RoboDK station: 4. Semi-Final Product.rdk

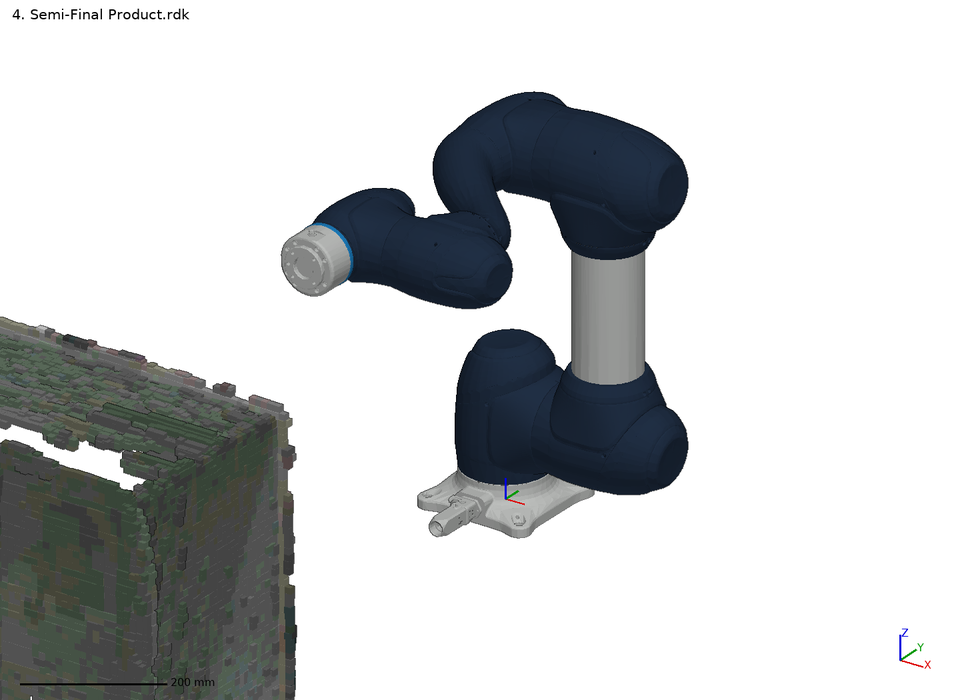
[picture v0: the station drawn from its stored meshes, robots at their saved joint values, targets as dots, program paths as lines]
Station Robotic 3D Mapping (saved by RoboDK 5.9.6). Poses are relative to the parent item; angles as X-Y-Z fixed-axis rotations.
  - frame Doosan Robotics M0609 Base at (0, 0, 0) mm
    - robot Doosan Robotics M0609: 6 axes, payload 6 kg, reach 900 mm, repeatability 0.03 mm, weight 27 kg
        modified DH rows (alpha deg, a mm, theta deg, d mm): 0, 0, 0, 135; -90, 0, -90, -6.207; 0, 411, -90, 0; -90, 0, 0, 368; 90, 0, 0, 0; -90, 0, 180, 121
        base shift (0, 0, 0) mm, rotated rx 0 ry 0 rz 180 deg
        joint limits [-360, -360, -150, -360, -360, -360] to [360, 360, 150, 360, 360, 360]; home [0, 0, 90, 0, 0, 0]; saved at [-90, 0, 90, 0, 0, 0]
      - tool Intel RealSense D455F, TCP at (0, 0, 0) mm
    - camera Camera 1
    - object Robot Base - Colored Cleaned Scan Mesh at (0, 0, 0) mm, size 1017.6 x 398.4 x 619.5 mm, geometry from 02_scan_cleaned_inside_stl_range_ROBODK_MM_COLORED.obj
  - Python program Prog1 (listed below)
  - Python program Prog2 (listed below)
  - Python program Prog3 (listed below)
  - Python program Prog4 (listed below)
  - Python program Prog5 (listed below)
  - Python program Prog6 (listed below)

--- Python program Prog1 ---
import sys
import time
from pathlib import Path

import numpy as np
import open3d as o3d
import pyrealsense2 as rs

sys.path.append("C:/RoboDK/Python")

from robodk.robolink import *
from robodk.robomath import TxyzRxyz_2_Pose, Mat


# ─────────────────────────────────────────────────────────────────────────────
# CONFIGURATION
# ─────────────────────────────────────────────────────────────────────────────

RUN_ON_REAL_ROBOT = True

HOME_JOINTS = [270.00, 0.00, 90.00, 180.00, 0.00, 0.00]

CENTER_REFERENCE_JOINTS = [270.01, 0.21, 98.95, 180.00, 6.92, 0.00]

TCP_TO_CAMERA_MOUNT = [0, 0, 55, 0, 0, 0]
CAMERA_MOUNT_TO_OPTICAL = [0, 0, 0, 0, 0, 90]

MIN_SAFE_TCP_Z_MM = 120.0
MIN_SAFE_CAMERA_Z_MM = 120.0

RS_WIDTH = 848
RS_HEIGHT = 480
RS_FPS = 30

WARMUP_FRAMES = 30
CAPTURE_FRAMES_PER_POSITION = 30

DEPTH_TRUNC_MAX = 1.0

SETTLE_TIME = 1.5
MOVE_TIMEOUT_SEC = 30.0
POLL_INTERVAL_SEC = 0.1

SURFACE_VOXEL_SIZE = 0.003

OUTLIER_NB_NEIGHBORS = 20
OUTLIER_STD_RATIO = 2.0

NORMAL_RADIUS = 0.02
NORMAL_MAX_NN = 30

SHOW_FINAL_CLOUD = True
SHOW_DEBUG_EACH_SCAN = False

MIN_SIDE_OFFSET_M = 0.08
MAX_SIDE_OFFSET_M = 0.32

MIN_VERTICAL_OFFSET_M = 0.06
MAX_VERTICAL_OFFSET_M = 0.24

MIN_FORWARD_OFFSET_M = 0.03
MAX_FORWARD_OFFSET_M = 0.14

ADAPTIVE_CROP_MARGIN_X_M = 0.12
ADAPTIVE_CROP_MARGIN_Y_M = 0.12
ADAPTIVE_CROP_MARGIN_Z_M = 0.20

BOUNDS_LOW_PERCENTILE = 2.0
BOUNDS_HIGH_PERCENTILE = 98.0

MIN_REFERENCE_POINTS = 1000

OUTPUT_FOLDER = Path(
    "C:/Users/daryl/Desktop/Robotic D Environment Mapping/"
    "Robotic-3D-Environment-Mapping/Point Cloud Testing Folder"
)

OUTPUT_CLEAN_FILE = OUTPUT_FOLDER / "adaptive_inside_box_pointcloud_clean.pcd"


# ─────────────────────────────────────────────────────────────────────────────
# ROBODK MATRIX HELPERS
# ─────────────────────────────────────────────────────────────────────────────

def robodk_mat_to_numpy(mat):
    transform = np.eye(4, dtype=np.float64)

    for row in range(3):
        for col in range(3):
            transform[row, col] = mat[row, col]

        transform[row, 3] = mat[row, 3] / 1000.0

    return transform


def numpy_to_robodk_mat(transform):
    return Mat([
        [
            transform[0, 0],
            transform[0, 1],
            transform[0, 2],
            transform[0, 3] * 1000.0,
        ],
        [
            transform[1, 0],
            transform[1, 1],
            transform[1, 2],
            transform[1, 3] * 1000.0,
        ],
        [
            transform[2, 0],
            transform[2, 1],
            transform[2, 2],
            transform[2, 3] * 1000.0,
        ],
        [0, 0, 0, 1],
    ])


def xyzrxryrz_to_numpy(pose_values):
    pose = TxyzRxyz_2_Pose([
        pose_values[0],
        pose_values[1],
        pose_values[2],
        np.radians(pose_values[3]),
        np.radians(pose_values[4]),
        np.radians(pose_values[5]),
    ])

    return robodk_mat_to_numpy(pose)


def make_local_offset_transform(offset_x, offset_y, offset_z):
    transform = np.eye(4, dtype=np.float64)
    transform[0, 3] = offset_x
    transform[1, 3] = offset_y
    transform[2, 3] = offset_z
    return transform


def joints_to_list(joints_mat):
    try:
        return list(joints_mat.list())
    except Exception:
        try:
            return list(joints_mat)
        except Exception:
            return [joints_mat[index] for index in range(len(joints_mat))]


def clamp(value, minimum_value, maximum_value):
    return max(minimum_value, min(value, maximum_value))


# ─────────────────────────────────────────────────────────────────────────────
# ROBODK ROBOT HELPERS
# ─────────────────────────────────────────────────────────────────────────────

def connect_robot(robot, rdk):
    if RUN_ON_REAL_ROBOT:
        rdk.setRunMode(RUNMODE_RUN_ROBOT)

        status = robot.ConnectSafe()
        print("ConnectSafe status:", status)

        if status != ROBOTCOM_READY:
            raise Exception("Robot is not ready. Check RoboDK connection settings.")
    else:
        rdk.setRunMode(RUNMODE_SIMULATE)
        print("Running in RoboDK simulation mode.")


def wait_until_robot_stops(robot, timeout_sec=MOVE_TIMEOUT_SEC):
    start = time.time()

    while True:
        try:
            if not robot.Busy():
                return
        except Exception:
            pass

        if time.time() - start > timeout_sec:
            raise Exception("Timeout waiting for robot to stop.")

        time.sleep(POLL_INTERVAL_SEC)


def get_robot_joints_when_ready(robot, timeout_sec=5.0):
    start = time.time()

    while True:
        try:
            return joints_to_list(robot.Joints())
        except Exception:
            if time.time() - start > timeout_sec:
                raise Exception("Could not read robot joints.")

            time.sleep(POLL_INTERVAL_SEC)


def move_robot_to_joints(robot, rdk, joints, label):
    target = rdk.AddTarget(f"_adaptive_inside_box_{label}")
    target.setAsJointTarget()
    target.setJoints(joints)

    print(f"\nMoving to {label}: {[round(joint, 2) for joint in joints]}")

    if RUN_ON_REAL_ROBOT:
        rdk.setRunMode(RUNMODE_RUN_ROBOT)
    else:
        rdk.setRunMode(RUNMODE_SIMULATE)

    robot.MoveJ(target, blocking=False)

    wait_until_robot_stops(robot)

    target.Delete()

    print(f"Arrived at {label}. Settling for {SETTLE_TIME:.1f} seconds...")
    time.sleep(SETTLE_TIME)

    return get_robot_joints_when_ready(robot)


def move_robot_to_pose(robot, rdk, T_base_tcp, label):
    target = rdk.AddTarget(f"_adaptive_inside_box_{label}")
    target_pose = numpy_to_robodk_mat(T_base_tcp)

    target.setPose(target_pose)
    target.setAsCartesianTarget()

    print(f"\nMoving to generated pose: {label}")
    print("Target TCP position in robot base frame:")
    print(f"X: {T_base_tcp[0, 3] * 1000.0:.1f} mm")
    print(f"Y: {T_base_tcp[1, 3] * 1000.0:.1f} mm")
    print(f"Z: {T_base_tcp[2, 3] * 1000.0:.1f} mm")

    if RUN_ON_REAL_ROBOT:
        rdk.setRunMode(RUNMODE_RUN_ROBOT)
    else:
        rdk.setRunMode(RUNMODE_SIMULATE)

    robot.MoveJ(target, blocking=False)

    wait_until_robot_stops(robot)

    target.Delete()

    print(f"Arrived at {label}. Settling for {SETTLE_TIME:.1f} seconds...")
    time.sleep(SETTLE_TIME)

    return get_robot_joints_when_ready(robot)


def is_generated_pose_safe(T_base_tcp, T_base_camera, label):
    tcp_z_mm = T_base_tcp[2, 3] * 1000.0
    camera_z_mm = T_base_camera[2, 3] * 1000.0

    if tcp_z_mm < MIN_SAFE_TCP_Z_MM:
        print("")
        print(f"SKIPPING {label}")
        print(f"Reason: TCP Z is too low: {tcp_z_mm:.1f} mm")
        print(f"Minimum safe TCP Z: {MIN_SAFE_TCP_Z_MM:.1f} mm")
        return False

    if camera_z_mm < MIN_SAFE_CAMERA_Z_MM:
        print("")
        print(f"SKIPPING {label}")
        print(f"Reason: Camera Z is too low: {camera_z_mm:.1f} mm")
        print(f"Minimum safe camera Z: {MIN_SAFE_CAMERA_Z_MM:.1f} mm")
        return False

    return True


def print_transform(name, transform):
    print(f"\n{name}:")
    print(np.round(transform, 6))


def print_cloud_bounds(name, point_cloud):
    if len(point_cloud.points) == 0:
        print(f"{name}: empty point cloud")
        return

    bounding_box = point_cloud.get_axis_aligned_bounding_box()

    print("")
    print(name)
    print("Points:", len(point_cloud.points))
    print("Min bound:", np.round(bounding_box.get_min_bound(), 4))
    print("Max bound:", np.round(bounding_box.get_max_bound(), 4))
    print("Center   :", np.round(bounding_box.get_center(), 4))
    print("Extent   :", np.round(bounding_box.get_extent(), 4))


# ─────────────────────────────────────────────────────────────────────────────
# REALSENSE HELPERS
# ─────────────────────────────────────────────────────────────────────────────

def start_realsense():
    print("\nStarting Intel RealSense D455f...")

    pipeline = rs.pipeline()
    config = rs.config()

    config.enable_stream(rs.stream.depth, RS_WIDTH, RS_HEIGHT, rs.format.z16, RS_FPS)
    config.enable_stream(rs.stream.color, RS_WIDTH, RS_HEIGHT, rs.format.rgb8, RS_FPS)

    profile = pipeline.start(config)

    depth_sensor = profile.get_device().first_depth_sensor()

    if depth_sensor.supports(rs.option.visual_preset):
        try:
            depth_sensor.set_option(
                rs.option.visual_preset,
                int(rs.rs400_visual_preset.high_density)
            )
            print("Visual preset: HIGH_DENSITY")
        except Exception as error:
            print("Could not set HIGH_DENSITY preset:", error)

    if depth_sensor.supports(rs.option.emitter_enabled):
        try:
            depth_sensor.set_option(rs.option.emitter_enabled, 1)
            print("Emitter enabled.")
        except Exception as error:
            print("Could not enable emitter:", error)

    if depth_sensor.supports(rs.option.laser_power):
        try:
            laser_range = depth_sensor.get_option_range(rs.option.laser_power)
            depth_sensor.set_option(rs.option.laser_power, laser_range.max)
            print("Laser power set to max:", laser_range.max)
        except Exception as error:
            print("Could not set laser power:", error)

    depth_scale = depth_sensor.get_depth_scale()
    print("Depth scale:", depth_scale)

    spatial_filter = rs.spatial_filter()
    temporal_filter = rs.temporal_filter()
    hole_filling_filter = rs.hole_filling_filter()

    spatial_filter.set_option(rs.option.filter_magnitude, 2)
    spatial_filter.set_option(rs.option.filter_smooth_alpha, 0.5)
    spatial_filter.set_option(rs.option.filter_smooth_delta, 20)

    hole_filling_filter.set_option(rs.option.holes_fill, 1)

    align = rs.align(rs.stream.color)

    print(f"Warming up RealSense for {WARMUP_FRAMES} frames...")
    for _ in range(WARMUP_FRAMES):
        pipeline.wait_for_frames()

    color_stream = profile.get_stream(rs.stream.color).as_video_stream_profile()
    intrinsics = color_stream.get_intrinsics()

    intrinsic_o3d = o3d.camera.PinholeCameraIntrinsic(
        intrinsics.width,
        intrinsics.height,
        intrinsics.fx,
        intrinsics.fy,
        intrinsics.ppx,
        intrinsics.ppy,
    )

    print(f"RealSense ready: fx={intrinsics.fx:.1f}, fy={intrinsics.fy:.1f}")

    return (
        pipeline,
        align,
        depth_scale,
        intrinsic_o3d,
        spatial_filter,
        temporal_filter,
        hole_filling_filter,
    )


def make_rgbd(color_image, depth_image, depth_scale_value):
    color_o3d = o3d.geometry.Image(color_image.astype(np.uint8))
    depth_o3d = o3d.geometry.Image(depth_image.astype(np.uint16))

    return o3d.geometry.RGBDImage.create_from_color_and_depth(
        color_o3d,
        depth_o3d,
        depth_scale=1.0 / depth_scale_value,
        depth_trunc=DEPTH_TRUNC_MAX,
        convert_rgb_to_intensity=False,
    )


def capture_stable_pointcloud(
    pipeline,
    align,
    intrinsic_o3d,
    depth_scale_value,
    spatial_filter,
    temporal_filter,
    hole_filling_filter,
    frames_to_capture=CAPTURE_FRAMES_PER_POSITION
):
    color_stack = []
    depth_stack = []

    print(f"Capturing {frames_to_capture} frames...")

    for frame_index in range(frames_to_capture):
        frames = pipeline.wait_for_frames()
        aligned_frames = align.process(frames)

        depth_frame = aligned_frames.get_depth_frame()
        color_frame = aligned_frames.get_color_frame()

        if not depth_frame or not color_frame:
            print(f"Frame {frame_index + 1}: skipped because depth or color is missing.")
            continue

        depth_frame = spatial_filter.process(depth_frame)
        depth_frame = temporal_filter.process(depth_frame)
        depth_frame = hole_filling_filter.process(depth_frame)

        depth_stack.append(np.asanyarray(depth_frame.get_data()).astype(np.uint16))
        color_stack.append(np.asanyarray(color_frame.get_data()).astype(np.uint8))

        print(f"Frame {frame_index + 1}/{frames_to_capture} captured.")

    if not depth_stack:
        return None

    print("Combining frames into one stable point cloud...")

    depth_median = np.median(np.stack(depth_stack, axis=0), axis=0).astype(np.uint16)
    color_mean = np.mean(np.stack(color_stack, axis=0), axis=0).astype(np.uint8)

    rgbd = make_rgbd(color_mean, depth_median, depth_scale_value)

    point_cloud = o3d.geometry.PointCloud.create_from_rgbd_image(
        rgbd,
        intrinsic_o3d,
    )

    if len(point_cloud.points) == 0:
        return None

    return point_cloud


# ─────────────────────────────────────────────────────────────────────────────
# ADAPTIVE POINT CLOUD HELPERS
# ─────────────────────────────────────────────────────────────────────────────

def estimate_camera_cloud_bounds(point_cloud):
    points = np.asarray(point_cloud.points)

    if len(points) < MIN_REFERENCE_POINTS:
        raise Exception(
            f"Not enough points for adaptive scan estimation. "
            f"Points found: {len(points)}"
        )

    valid_mask = (
        np.isfinite(points[:, 0]) &
        np.isfinite(points[:, 1]) &
        np.isfinite(points[:, 2]) &
        (points[:, 2] > 0.05) &
        (points[:, 2] < DEPTH_TRUNC_MAX)
    )

    points = points[valid_mask]

    if len(points) < MIN_REFERENCE_POINTS:
        raise Exception(
            f"Not enough valid depth points for adaptive scan estimation. "
            f"Valid points found: {len(points)}"
        )

    min_x = np.percentile(points[:, 0], BOUNDS_LOW_PERCENTILE)
    max_x = np.percentile(points[:, 0], BOUNDS_HIGH_PERCENTILE)

    min_y = np.percentile(points[:, 1], BOUNDS_LOW_PERCENTILE)
    max_y = np.percentile(points[:, 1], BOUNDS_HIGH_PERCENTILE)

    min_z = np.percentile(points[:, 2], BOUNDS_LOW_PERCENTILE)
    max_z = np.percentile(points[:, 2], BOUNDS_HIGH_PERCENTILE)

    center_x = float((min_x + max_x) / 2.0)
    center_y = float((min_y + max_y) / 2.0)
    center_z = float(np.median(points[:, 2]))

    extent_x = float(max_x - min_x)
    extent_y = float(max_y - min_y)
    extent_z = float(max_z - min_z)

    bounds = {
        "min_x": float(min_x),
        "max_x": float(max_x),
        "min_y": float(min_y),
        "max_y": float(max_y),
        "min_z": float(min_z),
        "max_z": float(max_z),
        "center_x": center_x,
        "center_y": center_y,
        "center_z": center_z,
        "extent_x": extent_x,
        "extent_y": extent_y,
        "extent_z": extent_z,
    }

    print("")
    print("Adaptive camera-frame bounds estimated from reference scan:")
    for key, value in bounds.items():
        print(f"{key}: {value:.4f} m")

    return bounds


def crop_pointcloud_adaptive(point_cloud, adaptive_bounds):
    if len(point_cloud.points) == 0:
        return point_cloud

    points = np.asarray(point_cloud.points)

    min_x = adaptive_bounds["min_x"] - ADAPTIVE_CROP_MARGIN_X_M
    max_x = adaptive_bounds["max_x"] + ADAPTIVE_CROP_MARGIN_X_M

    min_y = adaptive_bounds["min_y"] - ADAPTIVE_CROP_MARGIN_Y_M
    max_y = adaptive_bounds["max_y"] + ADAPTIVE_CROP_MARGIN_Y_M

    min_z = max(0.05, adaptive_bounds["min_z"] - ADAPTIVE_CROP_MARGIN_Z_M)
    max_z = min(DEPTH_TRUNC_MAX, adaptive_bounds["max_z"] + ADAPTIVE_CROP_MARGIN_Z_M)

    mask = (
        (points[:, 0] >= min_x) &
        (points[:, 0] <= max_x) &
        (points[:, 1] >= min_y) &
        (points[:, 1] <= max_y) &
        (points[:, 2] >= min_z) &
        (points[:, 2] <= max_z)
    )

    indices = np.where(mask)[0]

    if len(indices) == 0:
        print("WARNING: Adaptive crop removed all points. Keeping original cloud.")
        return point_cloud

    cropped_cloud = point_cloud.select_by_index(indices)

    print("Adaptive camera-frame crop enabled.")
    print("Points before adaptive crop:", len(point_cloud.points))
    print("Points after adaptive crop :", len(cropped_cloud.points))

    return cropped_cloud


def clean_pointcloud(point_cloud):
    if len(point_cloud.points) == 0:
        return point_cloud

    point_cloud = point_cloud.voxel_down_sample(voxel_size=SURFACE_VOXEL_SIZE)

    if len(point_cloud.points) == 0:
        return point_cloud

    point_cloud, _ = point_cloud.remove_statistical_outlier(
        nb_neighbors=OUTLIER_NB_NEIGHBORS,
        std_ratio=OUTLIER_STD_RATIO,
    )

    return point_cloud


def estimate_normals(point_cloud):
    if len(point_cloud.points) == 0:
        return point_cloud

    point_cloud.estimate_normals(
        search_param=o3d.geometry.KDTreeSearchParamHybrid(
            radius=NORMAL_RADIUS,
            max_nn=NORMAL_MAX_NN,
        )
    )

    return point_cloud


def save_debug_scan(label, point_cloud):
    debug_file = OUTPUT_FOLDER / f"debug_{label}.pcd"

    o3d.io.write_point_cloud(str(debug_file), point_cloud)

    print("Saved debug scan:", debug_file)
    print_cloud_bounds(f"Debug scan bounds - {label}", point_cloud)


# ─────────────────────────────────────────────────────────────────────────────
# ADAPTIVE SCAN POSE GENERATION
# ─────────────────────────────────────────────────────────────────────────────

def generate_adaptive_scan_offsets(adaptive_bounds):
    extent_x = adaptive_bounds["extent_x"]
    extent_y = adaptive_bounds["extent_y"]

    center_x = adaptive_bounds["center_x"]
    center_y = adaptive_bounds["center_y"]
    center_z = adaptive_bounds["center_z"]

    side_offset = clamp(
        extent_x * 0.35,
        MIN_SIDE_OFFSET_M,
        MAX_SIDE_OFFSET_M,
    )

    vertical_offset = clamp(
        extent_y * 0.35,
        MIN_VERTICAL_OFFSET_M,
        MAX_VERTICAL_OFFSET_M,
    )

    forward_offset = clamp(
        center_z * 0.12,
        MIN_FORWARD_OFFSET_M,
        MAX_FORWARD_OFFSET_M,
    )

    print("")
    print("Adaptive scan movement offsets:")
    print(f"Side offset: {side_offset:.4f} m")
    print(f"Vertical offset: {vertical_offset:.4f} m")
    print(f"Forward offset: {forward_offset:.4f} m")

    return [
        ("Reference_Center", 0.00, 0.00, 0.00),

        ("Left_Inside_Area", center_x - side_offset, center_y, 0.00),
        ("Right_Inside_Area", center_x + side_offset, center_y, 0.00),

        ("Upper_Inside_Area", center_x, center_y - vertical_offset, 0.00),
        ("Lower_Inside_Area", center_x, center_y + vertical_offset, 0.00),

        ("Upper_Left_Inside_Area", center_x - side_offset, center_y - vertical_offset, 0.00),
        ("Upper_Right_Inside_Area", center_x + side_offset, center_y - vertical_offset, 0.00),

        ("Lower_Left_Inside_Area", center_x - side_offset, center_y + vertical_offset, 0.00),
        ("Lower_Right_Inside_Area", center_x + side_offset, center_y + vertical_offset, 0.00),

        ("Closer_Center", center_x, center_y, forward_offset),
        ("Closer_Left", center_x - side_offset * 0.70, center_y, forward_offset),
        ("Closer_Right", center_x + side_offset * 0.70, center_y, forward_offset),
        ("Closer_Upper", center_x, center_y - vertical_offset * 0.70, forward_offset),
        ("Closer_Lower", center_x, center_y + vertical_offset * 0.70, forward_offset),
    ]


def generate_scan_camera_poses_from_center(T_base_camera_center, adaptive_bounds):
    generated_poses = []

    adaptive_offsets = generate_adaptive_scan_offsets(adaptive_bounds)

    print("\nGenerating adaptive scan poses from center reference...")
    print("Center camera position in robot base frame:")
    print(f"X: {T_base_camera_center[0, 3] * 1000.0:.1f} mm")
    print(f"Y: {T_base_camera_center[1, 3] * 1000.0:.1f} mm")
    print(f"Z: {T_base_camera_center[2, 3] * 1000.0:.1f} mm")

    for label, offset_x, offset_y, offset_z in adaptive_offsets:
        T_camera_offset = make_local_offset_transform(
            offset_x,
            offset_y,
            offset_z,
        )

        T_base_camera_target = T_base_camera_center @ T_camera_offset

        print("")
        print(f"Generated camera pose: {label}")
        print(f"Local offset X: {offset_x * 1000.0:.1f} mm")
        print(f"Local offset Y: {offset_y * 1000.0:.1f} mm")
        print(f"Local offset Z: {offset_z * 1000.0:.1f} mm")
        print("Generated camera position in robot base frame:")
        print(f"X: {T_base_camera_target[0, 3] * 1000.0:.1f} mm")
        print(f"Y: {T_base_camera_target[1, 3] * 1000.0:.1f} mm")
        print(f"Z: {T_base_camera_target[2, 3] * 1000.0:.1f} mm")

        generated_poses.append((label, T_base_camera_target))

    return generated_poses


# ─────────────────────────────────────────────────────────────────────────────
# SCANNING LOGIC
# ─────────────────────────────────────────────────────────────────────────────

def scan_current_position(
    label,
    pipeline,
    align,
    intrinsic_o3d,
    depth_scale,
    spatial_filter,
    temporal_filter,
    hole_filling_filter,
    T_base_camera_actual,
    adaptive_bounds=None,
):
    point_cloud = capture_stable_pointcloud(
        pipeline,
        align,
        intrinsic_o3d,
        depth_scale,
        spatial_filter,
        temporal_filter,
        hole_filling_filter,
        CAPTURE_FRAMES_PER_POSITION,
    )

    if point_cloud is None:
        print(f"WARNING: Empty point cloud at {label}.")
        return None

    print(f"Captured raw camera points at {label}: {len(point_cloud.points):,}")
    print_cloud_bounds(f"Raw camera-frame scan - {label}", point_cloud)

    if adaptive_bounds is not None:
        point_cloud = crop_pointcloud_adaptive(point_cloud, adaptive_bounds)

    if len(point_cloud.points) == 0:
        print(f"WARNING: Empty point cloud after adaptive crop at {label}.")
        return None

    print_cloud_bounds(f"Cropped camera-frame scan - {label}", point_cloud)

    point_cloud.transform(T_base_camera_actual)

    clean_scan = clean_pointcloud(point_cloud)

    if len(clean_scan.points) == 0:
        print(f"WARNING: Point cloud empty after cleaning at {label}.")
        return None

    save_debug_scan(label, clean_scan)

    if SHOW_DEBUG_EACH_SCAN:
        o3d.visualization.draw_geometries(
            [clean_scan],
            window_name=f"Debug transformed scan - {label}",
        )

    return clean_scan


# ─────────────────────────────────────────────────────────────────────────────
# MAIN
# ─────────────────────────────────────────────────────────────────────────────

def main():
    OUTPUT_FOLDER.mkdir(parents=True, exist_ok=True)

    rdk = Robolink()

    robot = rdk.ItemUserPick("Select your Doosan M0609 robot", ITEM_TYPE_ROBOT)

    if not robot.Valid():
        raise Exception("No valid robot selected.")

    print("Selected robot:", robot.Name())

    connect_robot(robot, rdk)

    T_tcp_mount = xyzrxryrz_to_numpy(TCP_TO_CAMERA_MOUNT)
    T_mount_optical = xyzrxryrz_to_numpy(CAMERA_MOUNT_TO_OPTICAL)
    T_tcp_camera = T_tcp_mount @ T_mount_optical
    T_camera_tcp = np.linalg.inv(T_tcp_camera)

    print_transform("T_tcp_camera", T_tcp_camera)

    pipeline = None
    combined_point_cloud = o3d.geometry.PointCloud()

    successful_scans = 0
    skipped_scans = 0
    unsafe_scans = 0
    failed_moves = 0

    try:
        move_robot_to_joints(
            robot,
            rdk,
            HOME_JOINTS,
            "Home_Start",
        )

        (
            pipeline,
            align,
            depth_scale,
            intrinsic_o3d,
            spatial_filter,
            temporal_filter,
            hole_filling_filter,
        ) = start_realsense()

        print("\n" + "=" * 70)
        print("ADAPTIVE INSIDE-BOX SCANNING STARTED")
        print("=" * 70)
        print("The robot moves to one manually taught center reference.")
        print("The first scan estimates the visible box size and distance.")
        print("The other scan poses are generated automatically from that estimate.")
        print("The code uses adaptive crop limits instead of a fixed 1 meter crop.")
        print("Generated poses below the robot-frame table safety limit are skipped.")
        print("=" * 70)

        center_actual_joints = move_robot_to_joints(
            robot,
            rdk,
            CENTER_REFERENCE_JOINTS,
            "Cabinet_Center_Reference",
        )

        T_base_tcp_center = robodk_mat_to_numpy(robot.SolveFK(center_actual_joints))
        T_base_camera_center = T_base_tcp_center @ T_tcp_camera

        print_transform("T_base_tcp_center", T_base_tcp_center)
        print_transform("T_base_camera_center", T_base_camera_center)

        reference_cloud = capture_stable_pointcloud(
            pipeline,
            align,
            intrinsic_o3d,
            depth_scale,
            spatial_filter,
            temporal_filter,
            hole_filling_filter,
            CAPTURE_FRAMES_PER_POSITION,
        )

        if reference_cloud is None:
            raise Exception("Reference scan failed. No point cloud was captured.")

        print_cloud_bounds("Reference raw camera-frame scan", reference_cloud)

        adaptive_bounds = estimate_camera_cloud_bounds(reference_cloud)

        reference_cloud_cropped = crop_pointcloud_adaptive(
            reference_cloud,
            adaptive_bounds,
        )

        reference_cloud_cropped.transform(T_base_camera_center)
        reference_clean_scan = clean_pointcloud(reference_cloud_cropped)

        if len(reference_clean_scan.points) > 0:
            save_debug_scan("Reference_Center", reference_clean_scan)
            combined_point_cloud += reference_clean_scan
            successful_scans += 1
            print(
                f"Accepted scan {successful_scans}: Reference_Center "
                f"with {len(reference_clean_scan.points):,} cleaned points"
            )
        else:
            print("WARNING: Reference scan became empty after cleaning.")
            skipped_scans += 1

        generated_camera_poses = generate_scan_camera_poses_from_center(
            T_base_camera_center,
            adaptive_bounds,
        )

        for label, T_base_camera_target in generated_camera_poses:
            if label == "Reference_Center":
                continue

            T_base_tcp_target = T_base_camera_target @ T_camera_tcp

            if not is_generated_pose_safe(
                T_base_tcp_target,
                T_base_camera_target,
                label,
            ):
                unsafe_scans += 1
                skipped_scans += 1
                continue

            try:
                actual_joints = move_robot_to_pose(
                    robot,
                    rdk,
                    T_base_tcp_target,
                    label,
                )
            except Exception as error:
                print("")
                print(f"WARNING: Could not move to generated pose {label}.")
                print("Move error:", error)
                failed_moves += 1
                skipped_scans += 1
                continue

            T_base_tcp_actual = robodk_mat_to_numpy(robot.SolveFK(actual_joints))
            T_base_camera_actual = T_base_tcp_actual @ T_tcp_camera

            print_transform(f"T_base_tcp_actual_{label}", T_base_tcp_actual)
            print_transform(f"T_base_camera_actual_{label}", T_base_camera_actual)

            clean_scan = scan_current_position(
                label,
                pipeline,
                align,
                intrinsic_o3d,
                depth_scale,
                spatial_filter,
                temporal_filter,
                hole_filling_filter,
                T_base_camera_actual,
                adaptive_bounds,
            )

            if clean_scan is None:
                skipped_scans += 1
                continue

            combined_point_cloud += clean_scan
            successful_scans += 1

            print(
                f"Accepted scan {successful_scans}: {label} "
                f"with {len(clean_scan.points):,} cleaned points"
            )

    except KeyboardInterrupt:
        print("\nScanning interrupted by user.")

    finally:
        if pipeline is not None:
            pipeline.stop()
            print("\nRealSense stopped.")

        try:
            move_robot_to_joints(
                robot,
                rdk,
                HOME_JOINTS,
                "Home_End",
            )
        except Exception as error:
            print("Could not move robot back to home position:", error)

    print("\n" + "=" * 70)
    print("SCAN SUMMARY")
    print("=" * 70)
    print("Successful scans:", successful_scans)
    print("Skipped scans:", skipped_scans)
    print("Unsafe skipped scans:", unsafe_scans)
    print("Failed robot moves:", failed_moves)
    print("Total merged points before final cleanup:", len(combined_point_cloud.points))
    print_cloud_bounds("Combined point cloud before final cleanup", combined_point_cloud)

    if len(combined_point_cloud.points) == 0:
        raise Exception("No valid point cloud was captured. Combined cloud is empty.")

    combined_point_cloud = clean_pointcloud(combined_point_cloud)
    combined_point_cloud = estimate_normals(combined_point_cloud)

    print("Total merged points after final cleanup:", len(combined_point_cloud.points))
    print_cloud_bounds("Combined point cloud after final cleanup", combined_point_cloud)

    o3d.io.write_point_cloud(str(OUTPUT_CLEAN_FILE), combined_point_cloud)
    print("Saved final merged point cloud to:", OUTPUT_CLEAN_FILE)

    if SHOW_FINAL_CLOUD:
        o3d.visualization.draw_geometries(
            [combined_point_cloud],
            window_name=f"Adaptive Inside Box Point Cloud - {successful_scans} scans",
        )

    print("Done.")


if __name__ == "__main__":
    main()

--- Python program Prog2 ---
import sys
from pathlib import Path

sys.path.append("C:/RoboDK/Python")

from robodk.robolink import *


ROBOTDK_EXPORT_FOLDER = Path(
    r"C:/Users/daryl/Desktop/Robotic D Environment Mapping/"
    r"Robotic-3D-Environment-Mapping/RoboDK Export"
)

COLORED_SCAN_OBJ_FILE = (
    ROBOTDK_EXPORT_FOLDER / "02_scan_cleaned_inside_stl_range_ROBODK_MM_COLORED.obj"
)

COLORED_SCAN_MTL_FILE = (
    ROBOTDK_EXPORT_FOLDER / "02_scan_cleaned_inside_stl_range_ROBODK_MM_COLORED.mtl"
)

COLORED_SCAN_PLY_FILE = (
    ROBOTDK_EXPORT_FOLDER / "02_scan_cleaned_inside_stl_range_ROBODK_MM_COLORED.ply"
)

ALIGNED_CAD_STL_FILE = (
    ROBOTDK_EXPORT_FOLDER / "04_aligned_cabinet_ROBODK_MM.stl"
)


def validate_file_exists(file_path):
    if not file_path.exists():
        raise FileNotFoundError(f"File not found: {file_path}")


def delete_existing_item(rdk, item_name):
    existing_item = rdk.Item(item_name)

    if existing_item.Valid():
        existing_item.Delete()


def import_file_to_robodk(rdk, file_path, item_name):
    validate_file_exists(file_path)

    item = rdk.AddFile(str(file_path))

    if not item.Valid():
        raise Exception(f"Could not import file into RoboDK: {file_path}")

    item.setName(item_name)
    item.setVisible(True)

    return item


def main():
    rdk = Robolink()

    scan_item_name = "Robot Base - Colored Cleaned Scan Mesh"
    cad_item_name = "Robot Base - Aligned Cabinet STL"

    delete_existing_item(rdk, scan_item_name)
    delete_existing_item(rdk, cad_item_name)

    if COLORED_SCAN_OBJ_FILE.exists():
        validate_file_exists(COLORED_SCAN_MTL_FILE)

        cleaned_scan = import_file_to_robodk(
            rdk,
            COLORED_SCAN_OBJ_FILE,
            scan_item_name
        )

        imported_scan_file = COLORED_SCAN_OBJ_FILE

    elif COLORED_SCAN_PLY_FILE.exists():
        cleaned_scan = import_file_to_robodk(
            rdk,
            COLORED_SCAN_PLY_FILE,
            scan_item_name
        )

        imported_scan_file = COLORED_SCAN_PLY_FILE

    else:
        raise FileNotFoundError(
            "No colored scan file found. Expected OBJ or PLY:\n"
            f"{COLORED_SCAN_OBJ_FILE}\n"
            f"{COLORED_SCAN_PLY_FILE}"
        )

    aligned_cad = import_file_to_robodk(
        rdk,
        ALIGNED_CAD_STL_FILE,
        cad_item_name
    )

    aligned_cad.setColor([1.0, 0.0, 0.0, 0.35])

    print("")
    print("=" * 70)
    print("IMPORTED INTO ROBODK")
    print("=" * 70)
    print("Colored scan:", cleaned_scan.Name())
    print("Scan file   :", imported_scan_file)
    print("")
    print("Aligned CAD :", aligned_cad.Name())
    print("CAD file    :", ALIGNED_CAD_STL_FILE)
    print("")
    print("The colored scan should keep its scanned color if RoboDK reads the OBJ/MTL material.")
    print("The CAD model is imported as transparent red.")
    print("Both files are already scaled to millimeters.")
    print("They should appear in the robot base coordinate position.")


if __name__ == "__main__":
    main()

--- Python program Prog3 ---
import sys
import time

import numpy as np

sys.path.append("C:/RoboDK/Python")

from robodk.robolink import *
from robodk.robomath import TxyzRxyz_2_Pose, Mat


# ─────────────────────────────────────────────────────────────────────────────
# CONFIGURATION
# ─────────────────────────────────────────────────────────────────────────────

RUN_ON_REAL_ROBOT = True

HOME_JOINTS = [270.00, 0.00, 90.00, 180.00, 0.00, 0.00]

# Your safe center camera view.
CENTER_REFERENCE_JOINTS = [270.01, 0.21, 98.95, 180.00, 6.92, 0.00]

# Your confirmed calibration. Do not change.
TCP_TO_CAMERA_MOUNT = [0, 0, 55, 0, 0, 0]
CAMERA_MOUNT_TO_OPTICAL = [0, 0, 0, 0, 0, 90]

MIN_SAFE_TCP_Z_MM = 120.0
MIN_SAFE_CAMERA_Z_MM = 120.0

SETTLE_TIME = 1.5
MOVE_TIMEOUT_SEC = 30.0
POLL_INTERVAL_SEC = 0.1

# This controls the virtual line the camera will look at.
# Think of this as the edge line inside the camera view.
#
# X = left/right in camera frame
# Y = up/down in camera frame
# Z = forward/depth in camera frame
#
# If the robot looks too far left/right, reduce LINE_HALF_WIDTH_M.
# If it looks too high/low, adjust LINE_Y_M.
# If it looks too close/far, adjust LINE_Z_M.
LINE_HALF_WIDTH_M = 0.22
LINE_Y_M = 0.06
LINE_Z_M = 0.55

# Number of look poses from left corner → center → right corner.
NUM_LOOK_POINTS = 7

# Optional small camera position offset.
# Keep these 0 first.
CAMERA_FIXED_X_OFFSET_M = 0.0
CAMERA_FIXED_Y_OFFSET_M = 0.0
CAMERA_FIXED_Z_OFFSET_M = 0.0

CREATE_DEBUG_TARGETS = True


# ─────────────────────────────────────────────────────────────────────────────
# ROBODK MATRIX HELPERS
# ─────────────────────────────────────────────────────────────────────────────

def robodk_mat_to_numpy(mat):
    transform = np.eye(4, dtype=np.float64)

    for row in range(3):
        for col in range(3):
            transform[row, col] = mat[row, col]

        transform[row, 3] = mat[row, 3] / 1000.0

    return transform


def numpy_to_robodk_mat(transform):
    return Mat([
        [
            transform[0, 0],
            transform[0, 1],
            transform[0, 2],
            transform[0, 3] * 1000.0,
        ],
        [
            transform[1, 0],
            transform[1, 1],
            transform[1, 2],
            transform[1, 3] * 1000.0,
        ],
        [
            transform[2, 0],
            transform[2, 1],
            transform[2, 2],
            transform[2, 3] * 1000.0,
        ],
        [0, 0, 0, 1],
    ])


def xyzrxryrz_to_numpy(pose_values):
    pose = TxyzRxyz_2_Pose([
        pose_values[0],
        pose_values[1],
        pose_values[2],
        np.radians(pose_values[3]),
        np.radians(pose_values[4]),
        np.radians(pose_values[5]),
    ])

    return robodk_mat_to_numpy(pose)


def joints_to_list(joints_mat):
    try:
        return list(joints_mat.list())
    except Exception:
        try:
            return list(joints_mat)
        except Exception:
            return [joints_mat[index] for index in range(len(joints_mat))]


def normalize(vector):
    norm = np.linalg.norm(vector)

    if norm < 1e-9:
        raise Exception("Cannot normalize zero-length vector.")

    return vector / norm


def print_transform(name, transform):
    print(f"\n{name}:")
    print(np.round(transform, 6))


# ─────────────────────────────────────────────────────────────────────────────
# ROBODK ROBOT HELPERS
# ─────────────────────────────────────────────────────────────────────────────

def connect_robot(robot, rdk):
    if RUN_ON_REAL_ROBOT:
        rdk.setRunMode(RUNMODE_RUN_ROBOT)

        status = robot.ConnectSafe()
        print("ConnectSafe status:", status)

        if status != ROBOTCOM_READY:
            raise Exception("Robot is not ready. Check RoboDK connection settings.")
    else:
        rdk.setRunMode(RUNMODE_SIMULATE)
        print("Running in RoboDK simulation mode.")


def wait_until_robot_stops(robot, timeout_sec=MOVE_TIMEOUT_SEC):
    start = time.time()

    while True:
        try:
            if not robot.Busy():
                return
        except Exception:
            pass

        if time.time() - start > timeout_sec:
            raise Exception("Timeout waiting for robot to stop.")

        time.sleep(POLL_INTERVAL_SEC)


def get_robot_joints_when_ready(robot, timeout_sec=5.0):
    start = time.time()

    while True:
        try:
            return joints_to_list(robot.Joints())
        except Exception:
            if time.time() - start > timeout_sec:
                raise Exception("Could not read robot joints.")

            time.sleep(POLL_INTERVAL_SEC)


def move_robot_to_joints(robot, rdk, joints, label):
    target = rdk.AddTarget(f"_camera_neck_follow_{label}")
    target.setAsJointTarget()
    target.setJoints(joints)

    print(f"\nMoving to {label}: {[round(joint, 2) for joint in joints]}")

    if RUN_ON_REAL_ROBOT:
        rdk.setRunMode(RUNMODE_RUN_ROBOT)
    else:
        rdk.setRunMode(RUNMODE_SIMULATE)

    robot.MoveJ(target, blocking=False)

    wait_until_robot_stops(robot)

    target.Delete()

    print(f"Arrived at {label}. Settling for {SETTLE_TIME:.1f} seconds...")
    time.sleep(SETTLE_TIME)

    return get_robot_joints_when_ready(robot)


def move_robot_to_pose(robot, rdk, T_base_tcp, label):
    target = rdk.AddTarget(f"_camera_neck_follow_{label}")
    target_pose = numpy_to_robodk_mat(T_base_tcp)

    target.setPose(target_pose)
    target.setAsCartesianTarget()

    print(f"\nMoving to camera neck pose: {label}")
    print("Target TCP position in robot base frame:")
    print(f"X: {T_base_tcp[0, 3] * 1000.0:.1f} mm")
    print(f"Y: {T_base_tcp[1, 3] * 1000.0:.1f} mm")
    print(f"Z: {T_base_tcp[2, 3] * 1000.0:.1f} mm")

    if RUN_ON_REAL_ROBOT:
        rdk.setRunMode(RUNMODE_RUN_ROBOT)
    else:
        rdk.setRunMode(RUNMODE_SIMULATE)

    robot.MoveJ(target, blocking=False)

    wait_until_robot_stops(robot)

    target.Delete()

    print(f"Arrived at {label}. Settling for {SETTLE_TIME:.1f} seconds...")
    time.sleep(SETTLE_TIME)

    return get_robot_joints_when_ready(robot)


def is_generated_pose_safe(T_base_tcp, T_base_camera, label):
    tcp_z_mm = T_base_tcp[2, 3] * 1000.0
    camera_z_mm = T_base_camera[2, 3] * 1000.0

    if tcp_z_mm < MIN_SAFE_TCP_Z_MM:
        print("")
        print(f"SKIPPING {label}")
        print(f"Reason: TCP Z is too low: {tcp_z_mm:.1f} mm")
        print(f"Minimum safe TCP Z: {MIN_SAFE_TCP_Z_MM:.1f} mm")
        return False

    if camera_z_mm < MIN_SAFE_CAMERA_Z_MM:
        print("")
        print(f"SKIPPING {label}")
        print(f"Reason: Camera Z is too low: {camera_z_mm:.1f} mm")
        print(f"Minimum safe camera Z: {MIN_SAFE_CAMERA_Z_MM:.1f} mm")
        return False

    return True


# ─────────────────────────────────────────────────────────────────────────────
# CAMERA LOOK / NECK MOVEMENT LOGIC
# ─────────────────────────────────────────────────────────────────────────────

def transform_point(T, point):
    point_h = np.array(
        [point[0], point[1], point[2], 1.0],
        dtype=np.float64
    )

    transformed = T @ point_h

    return transformed[:3]


def get_fixed_camera_position(T_base_camera_center):
    camera_position = T_base_camera_center[:3, 3].copy()

    camera_position += np.array([
        CAMERA_FIXED_X_OFFSET_M,
        CAMERA_FIXED_Y_OFFSET_M,
        CAMERA_FIXED_Z_OFFSET_M,
    ], dtype=np.float64)

    return camera_position


def generate_camera_frame_line_points():
    left_corner = np.array(
        [-LINE_HALF_WIDTH_M, LINE_Y_M, LINE_Z_M],
        dtype=np.float64
    )

    edge_center = np.array(
        [0.0, LINE_Y_M, LINE_Z_M],
        dtype=np.float64
    )

    right_corner = np.array(
        [LINE_HALF_WIDTH_M, LINE_Y_M, LINE_Z_M],
        dtype=np.float64
    )

    left_count = NUM_LOOK_POINTS // 2 + 1
    right_count = NUM_LOOK_POINTS - left_count + 1

    left_to_center = np.linspace(
        left_corner,
        edge_center,
        left_count
    )

    center_to_right = np.linspace(
        edge_center,
        right_corner,
        right_count
    )[1:]

    points = np.vstack((left_to_center, center_to_right))

    print("")
    print("=" * 70)
    print("Generated camera-frame look line")
    print("=" * 70)
    print("Left corner :", np.round(left_corner, 4))
    print("Edge center :", np.round(edge_center, 4))
    print("Right corner:", np.round(right_corner, 4))

    for index, point in enumerate(points, start=1):
        print(f"Look point {index:02d}: {np.round(point, 4)} m")

    return points


def transform_look_points_to_base(T_base_camera_center, camera_frame_points):
    base_points = []

    for point in camera_frame_points:
        base_point = transform_point(
            T_base_camera_center,
            point
        )

        base_points.append(base_point)

    return base_points


def build_camera_look_at_pose(
    T_base_camera_reference,
    camera_position_base,
    look_at_point_base
):
    direction = look_at_point_base - camera_position_base
    camera_forward = normalize(direction)

    reference_rotation = T_base_camera_reference[:3, :3]

    reference_up = reference_rotation[:, 1]
    reference_right = reference_rotation[:, 0]

    camera_right = np.cross(reference_up, camera_forward)

    if np.linalg.norm(camera_right) < 1e-6:
        camera_right = reference_right
    else:
        camera_right = normalize(camera_right)

    camera_up = np.cross(camera_forward, camera_right)
    camera_up = normalize(camera_up)

    camera_right = np.cross(camera_up, camera_forward)
    camera_right = normalize(camera_right)

    T_base_camera = np.eye(4, dtype=np.float64)

    T_base_camera[:3, 0] = camera_right
    T_base_camera[:3, 1] = camera_up
    T_base_camera[:3, 2] = camera_forward
    T_base_camera[:3, 3] = camera_position_base

    return T_base_camera


# ─────────────────────────────────────────────────────────────────────────────
# ROBODK DEBUG TARGETS
# ─────────────────────────────────────────────────────────────────────────────

def delete_existing_item(rdk, name, item_type):
    item = rdk.Item(name, item_type)

    if item.Valid():
        item.Delete()


def create_target_marker(rdk, name, T_base_target):
    delete_existing_item(rdk, name, ITEM_TYPE_TARGET)

    target = rdk.AddTarget(name)
    target.setPose(numpy_to_robodk_mat(T_base_target))

    return target


def create_point_marker(rdk, name, position_base):
    T_base_target = np.eye(4, dtype=np.float64)
    T_base_target[:3, 3] = position_base

    return create_target_marker(
        rdk,
        name,
        T_base_target
    )


def create_debug_targets(
    rdk,
    look_points_base,
    camera_position_base,
    camera_pose_targets
):
    if not CREATE_DEBUG_TARGETS:
        return

    create_point_marker(
        rdk,
        "NECK_CAMERA_FIXED_POSITION",
        camera_position_base
    )

    for index, look_point in enumerate(look_points_base, start=1):
        create_point_marker(
            rdk,
            f"NECK_LOOK_POINT_{index:02d}",
            look_point
        )

    for index, T_base_tcp in enumerate(camera_pose_targets, start=1):
        create_target_marker(
            rdk,
            f"NECK_TCP_TARGET_{index:02d}",
            T_base_tcp
        )


# ─────────────────────────────────────────────────────────────────────────────
# MAIN
# ─────────────────────────────────────────────────────────────────────────────

def main():
    rdk = Robolink()

    robot = rdk.ItemUserPick(
        "Select your Doosan M0609 robot",
        ITEM_TYPE_ROBOT
    )

    if not robot.Valid():
        raise Exception("No valid robot selected.")

    print("Selected robot:", robot.Name())

    connect_robot(robot, rdk)

    T_tcp_mount = xyzrxryrz_to_numpy(TCP_TO_CAMERA_MOUNT)
    T_mount_optical = xyzrxryrz_to_numpy(CAMERA_MOUNT_TO_OPTICAL)

    T_tcp_camera = T_tcp_mount @ T_mount_optical
    T_camera_tcp = np.linalg.inv(T_tcp_camera)

    print_transform("T_tcp_camera", T_tcp_camera)

    try:
        move_robot_to_joints(
            robot,
            rdk,
            HOME_JOINTS,
            "Home_Start"
        )

        center_actual_joints = move_robot_to_joints(
            robot,
            rdk,
            CENTER_REFERENCE_JOINTS,
            "Center_Reference_View"
        )

        T_base_tcp_center = robodk_mat_to_numpy(
            robot.SolveFK(center_actual_joints)
        )

        T_base_camera_center = T_base_tcp_center @ T_tcp_camera

        print_transform("T_base_tcp_center", T_base_tcp_center)
        print_transform("T_base_camera_center", T_base_camera_center)

        camera_frame_look_points = generate_camera_frame_line_points()

        look_points_base = transform_look_points_to_base(
            T_base_camera_center,
            camera_frame_look_points
        )

        fixed_camera_position_base = get_fixed_camera_position(
            T_base_camera_center
        )

        camera_pose_targets = []

        print("")
        print("=" * 70)
        print("GENERATING CAMERA NECK FOLLOW POSES")
        print("=" * 70)
        print("Camera position stays fixed.")
        print("Only the camera orientation changes.")
        print("Motion: left corner → edge center → right corner.")
        print("=" * 70)

        for index, look_point_base in enumerate(look_points_base, start=1):
            label = f"Neck_Follow_Point_{index:02d}"

            print("")
            print(label)
            print("Camera fixed position:")
            print(np.round(fixed_camera_position_base * 1000.0, 2), "mm")
            print("Looking at:")
            print(np.round(look_point_base * 1000.0, 2), "mm")

            T_base_camera_look = build_camera_look_at_pose(
                T_base_camera_center,
                fixed_camera_position_base,
                look_point_base
            )

            T_base_tcp_look = T_base_camera_look @ T_camera_tcp

            camera_pose_targets.append(T_base_tcp_look)

            if not is_generated_pose_safe(
                T_base_tcp_look,
                T_base_camera_look,
                label
            ):
                continue

        create_debug_targets(
            rdk,
            look_points_base,
            fixed_camera_position_base,
            camera_pose_targets
        )

        print("")
        print("=" * 70)
        print("CAMERA NECK FOLLOW START")
        print("=" * 70)

        for index, T_base_tcp_target in enumerate(camera_pose_targets, start=1):
            label = f"Neck_Follow_Point_{index:02d}"

            move_robot_to_pose(
                robot,
                rdk,
                T_base_tcp_target,
                label
            )

        print("")
        print("=" * 70)
        print("CAMERA NECK FOLLOW FINISHED")
        print("=" * 70)

    except KeyboardInterrupt:
        print("")
        print("Movement interrupted by user.")

    finally:
        try:
            move_robot_to_joints(
                robot,
                rdk,
                HOME_JOINTS,
                "Home_End"
            )
        except Exception as error:
            print("Could not move robot back to home position:", error)

    print("Done.")


if __name__ == "__main__":
    main()

--- Python program Prog4 ---
import sys
import time

import numpy as np

sys.path.append("C:/RoboDK/Python")

from robodk.robolink import *
from robodk.robomath import TxyzRxyz_2_Pose, Mat


# ─────────────────────────────────────────────────────────────────────────────
# CONFIGURATION
# ─────────────────────────────────────────────────────────────────────────────

RUN_ON_REAL_ROBOT = True

HOME_JOINTS = [270.00, 0.00, 90.00, 180.00, 0.00, 0.00]

CENTER_REFERENCE_JOINTS = [270.01, 0.21, 98.95, 180.00, 6.92, 0.00]

# Existing sensor/camera calibration.
TCP_TO_CAMERA_MOUNT = [0, 0, 55, 0, 0, 0]
CAMERA_MOUNT_TO_OPTICAL = [0, 0, 0, 0, 0, 90]

MIN_SAFE_TCP_Z_MM = 120.0

SETTLE_TIME = 1.5
MOVE_TIMEOUT_SEC = 30.0
POLL_INTERVAL_SEC = 0.1

# The seam is defined in the camera frame.
# X = left/right
# Y = up/down
# Z = forward/depth
#
# Previous values were too far. These are closer and safer.
SEAM_HALF_WIDTH_M = 0.08
SEAM_Y_M = 0.06
SEAM_Z_M = 0.18

# Keeps the dry-run tip slightly above the imagined seam.
DRY_RUN_HEIGHT_OFFSET_M = 0.03

# Distance before the seam along the torch direction.
# Smaller = tip gets nearer to the edge.
TIP_STANDOFF_M = 0.02

NUM_PATH_POINTS = 5

# Keep J6 close to the center value, but allow RoboDK to solve IK.
LOCK_J6_WITH_SEED = True
MAX_J6_WARNING_DEGREES = 5.0

CREATE_DEBUG_TARGETS = True


# ─────────────────────────────────────────────────────────────────────────────
# MATRIX HELPERS
# ─────────────────────────────────────────────────────────────────────────────

def robodk_mat_to_numpy(mat):
    transform = np.eye(4, dtype=np.float64)

    for row in range(3):
        for col in range(3):
            transform[row, col] = mat[row, col]

        transform[row, 3] = mat[row, 3] / 1000.0

    return transform


def numpy_to_robodk_mat(transform):
    return Mat([
        [
            transform[0, 0],
            transform[0, 1],
            transform[0, 2],
            transform[0, 3] * 1000.0,
        ],
        [
            transform[1, 0],
            transform[1, 1],
            transform[1, 2],
            transform[1, 3] * 1000.0,
        ],
        [
            transform[2, 0],
            transform[2, 1],
            transform[2, 2],
            transform[2, 3] * 1000.0,
        ],
        [0, 0, 0, 1],
    ])


def xyzrxryrz_to_numpy(pose_values):
    pose = TxyzRxyz_2_Pose([
        pose_values[0],
        pose_values[1],
        pose_values[2],
        np.radians(pose_values[3]),
        np.radians(pose_values[4]),
        np.radians(pose_values[5]),
    ])

    return robodk_mat_to_numpy(pose)


def joints_to_list(joints_mat):
    try:
        return list(joints_mat.list())
    except Exception:
        try:
            return list(joints_mat)
        except Exception:
            return [joints_mat[index] for index in range(len(joints_mat))]


def normalize(vector):
    norm = np.linalg.norm(vector)

    if norm < 1e-9:
        raise Exception("Cannot normalize zero-length vector.")

    return vector / norm


def transform_point(transform, point):
    point_h = np.array(
        [point[0], point[1], point[2], 1.0],
        dtype=np.float64
    )

    transformed = transform @ point_h

    return transformed[:3]


def print_transform(name, transform):
    print(f"\n{name}:")
    print(np.round(transform, 6))


# ─────────────────────────────────────────────────────────────────────────────
# ROBOT HELPERS
# ─────────────────────────────────────────────────────────────────────────────

def connect_robot(robot, rdk):
    if RUN_ON_REAL_ROBOT:
        rdk.setRunMode(RUNMODE_RUN_ROBOT)

        status = robot.ConnectSafe()
        print("ConnectSafe status:", status)

        if status != ROBOTCOM_READY:
            raise Exception("Robot is not ready. Check RoboDK connection settings.")
    else:
        rdk.setRunMode(RUNMODE_SIMULATE)
        print("Running in RoboDK simulation mode.")


def wait_until_robot_stops(robot, timeout_sec=MOVE_TIMEOUT_SEC):
    start = time.time()

    while True:
        try:
            if not robot.Busy():
                return
        except Exception:
            pass

        if time.time() - start > timeout_sec:
            raise Exception("Timeout waiting for robot to stop.")

        time.sleep(POLL_INTERVAL_SEC)


def get_robot_joints_when_ready(robot, timeout_sec=5.0):
    start = time.time()

    while True:
        try:
            return joints_to_list(robot.Joints())
        except Exception:
            if time.time() - start > timeout_sec:
                raise Exception("Could not read robot joints.")

            time.sleep(POLL_INTERVAL_SEC)


def move_robot_to_joints(robot, rdk, joints, label):
    target = rdk.AddTarget(f"_angled_tip_path_{label}")
    target.setAsJointTarget()
    target.setJoints(joints)

    print(f"\nMoving to {label}: {[round(joint, 2) for joint in joints]}")

    if RUN_ON_REAL_ROBOT:
        rdk.setRunMode(RUNMODE_RUN_ROBOT)
    else:
        rdk.setRunMode(RUNMODE_SIMULATE)

    robot.MoveJ(target, blocking=False)

    wait_until_robot_stops(robot)

    target.Delete()

    print(f"Arrived at {label}. Settling for {SETTLE_TIME:.1f} seconds...")
    time.sleep(SETTLE_TIME)

    return get_robot_joints_when_ready(robot)


def move_robot_to_pose(
    robot,
    rdk,
    T_base_tcp,
    seed_joints,
    locked_j6_value,
    label
):
    target = rdk.AddTarget(f"_angled_tip_path_{label}")
    target_pose = numpy_to_robodk_mat(T_base_tcp)

    target.setPose(target_pose)
    target.setAsCartesianTarget()

    seed = list(seed_joints)

    if LOCK_J6_WITH_SEED:
        seed[5] = locked_j6_value

    target.setJoints(seed)

    print(f"\nMoving to angled tip pose: {label}")
    print("Target TCP position in robot base frame:")
    print(f"X: {T_base_tcp[0, 3] * 1000.0:.1f} mm")
    print(f"Y: {T_base_tcp[1, 3] * 1000.0:.1f} mm")
    print(f"Z: {T_base_tcp[2, 3] * 1000.0:.1f} mm")
    print("Seed joints:")
    print([round(joint, 2) for joint in seed])

    if RUN_ON_REAL_ROBOT:
        rdk.setRunMode(RUNMODE_RUN_ROBOT)
    else:
        rdk.setRunMode(RUNMODE_SIMULATE)

    robot.MoveJ(target, blocking=False)

    wait_until_robot_stops(robot)

    actual_joints = get_robot_joints_when_ready(robot)

    target.Delete()

    print(f"Arrived at {label}. Settling for {SETTLE_TIME:.1f} seconds...")
    print("Actual joints:")
    print([round(joint, 2) for joint in actual_joints])
    print("Actual J6:", round(actual_joints[5], 2))

    if abs(actual_joints[5] - locked_j6_value) > MAX_J6_WARNING_DEGREES:
        print("")
        print("WARNING: J6 changed more than expected.")
        print("The angle may require a different wrist configuration.")

    time.sleep(SETTLE_TIME)

    return actual_joints


def is_pose_safe(T_base_tcp, label):
    tcp_z_mm = T_base_tcp[2, 3] * 1000.0

    if tcp_z_mm < MIN_SAFE_TCP_Z_MM:
        print("")
        print(f"SKIPPING {label}")
        print(f"Reason: TCP Z is too low: {tcp_z_mm:.1f} mm")
        return False

    return True


# ─────────────────────────────────────────────────────────────────────────────
# SEAM PATH GENERATION
# ─────────────────────────────────────────────────────────────────────────────

def generate_seam_points_camera_frame():
    left_corner = np.array(
        [
            -SEAM_HALF_WIDTH_M,
            SEAM_Y_M + DRY_RUN_HEIGHT_OFFSET_M,
            SEAM_Z_M
        ],
        dtype=np.float64
    )

    center_edge = np.array(
        [
            0.0,
            SEAM_Y_M + DRY_RUN_HEIGHT_OFFSET_M,
            SEAM_Z_M
        ],
        dtype=np.float64
    )

    right_corner = np.array(
        [
            SEAM_HALF_WIDTH_M,
            SEAM_Y_M + DRY_RUN_HEIGHT_OFFSET_M,
            SEAM_Z_M
        ],
        dtype=np.float64
    )

    left_count = NUM_PATH_POINTS // 2 + 1
    right_count = NUM_PATH_POINTS - left_count + 1

    left_to_center = np.linspace(
        left_corner,
        center_edge,
        left_count
    )

    center_to_right = np.linspace(
        center_edge,
        right_corner,
        right_count
    )[1:]

    points = np.vstack((left_to_center, center_to_right))

    print("")
    print("=" * 70)
    print("Generated angled seam points in camera frame")
    print("=" * 70)
    print("Left corner :", np.round(left_corner, 4))
    print("Center edge :", np.round(center_edge, 4))
    print("Right corner:", np.round(right_corner, 4))

    for index, point in enumerate(points, start=1):
        print(f"Seam point {index:02d}: {np.round(point, 4)} m")

    return points


def transform_seam_points_to_base(T_base_camera_center, seam_points_camera):
    seam_points_base = []

    for point in seam_points_camera:
        seam_points_base.append(
            transform_point(
                T_base_camera_center,
                point
            )
        )

    return seam_points_base


# ─────────────────────────────────────────────────────────────────────────────
# ANGLED TOOL FRAME
# ─────────────────────────────────────────────────────────────────────────────

def build_angled_tcp_pose(
    camera_position_base,
    seam_point_base,
    seam_direction_base,
    reference_rotation
):
    # Tool points from robot/camera side toward the seam.
    # This is the missing "angle where it is looking at".
    approach_axis = normalize(seam_point_base - camera_position_base)

    # Keep X roughly along the welding seam.
    tool_x_axis = seam_direction_base - np.dot(seam_direction_base, approach_axis) * approach_axis

    if np.linalg.norm(tool_x_axis) < 1e-6:
        tool_x_axis = reference_rotation[:, 0]
    else:
        tool_x_axis = normalize(tool_x_axis)

    # Build a clean right-handed orientation.
    tool_y_axis = np.cross(approach_axis, tool_x_axis)
    tool_y_axis = normalize(tool_y_axis)

    tool_x_axis = np.cross(tool_y_axis, approach_axis)
    tool_x_axis = normalize(tool_x_axis)

    # Keep the TCP slightly before the seam, so the tip is close but not too far in.
    tcp_position = seam_point_base - approach_axis * TIP_STANDOFF_M

    T_base_tcp = np.eye(4, dtype=np.float64)
    T_base_tcp[:3, 0] = tool_x_axis
    T_base_tcp[:3, 1] = tool_y_axis
    T_base_tcp[:3, 2] = approach_axis
    T_base_tcp[:3, 3] = tcp_position

    return T_base_tcp


def generate_angled_tcp_targets(
    T_base_camera_center,
    seam_points_base
):
    if len(seam_points_base) < 2:
        raise Exception("Not enough seam points.")

    camera_position_base = T_base_camera_center[:3, 3]
    reference_rotation = T_base_camera_center[:3, :3]

    seam_direction_base = seam_points_base[-1] - seam_points_base[0]
    seam_direction_base = normalize(seam_direction_base)

    targets = []

    print("")
    print("=" * 70)
    print("Generating angled TCP targets")
    print("=" * 70)
    print("The tool now points toward the seam.")
    print("The tip is closer because of TIP_STANDOFF_M.")

    for index, seam_point_base in enumerate(seam_points_base, start=1):
        label = f"Angled_Tip_Point_{index:02d}"

        T_base_tcp = build_angled_tcp_pose(
            camera_position_base,
            seam_point_base,
            seam_direction_base,
            reference_rotation
        )

        targets.append(
            (
                label,
                T_base_tcp,
                seam_point_base
            )
        )

        print("")
        print(label)
        print("Seam point:")
        print(np.round(seam_point_base * 1000.0, 2), "mm")
        print("TCP point:")
        print(np.round(T_base_tcp[:3, 3] * 1000.0, 2), "mm")
        print("Tool approach direction:")
        print(np.round(T_base_tcp[:3, 2], 4))

    return targets


# ─────────────────────────────────────────────────────────────────────────────
# DEBUG TARGETS
# ─────────────────────────────────────────────────────────────────────────────

def delete_existing_item(rdk, name, item_type):
    item = rdk.Item(name, item_type)

    if item.Valid():
        item.Delete()


def create_target_marker(rdk, name, T_base_target):
    if not CREATE_DEBUG_TARGETS:
        return None

    delete_existing_item(rdk, name, ITEM_TYPE_TARGET)

    target = rdk.AddTarget(name)
    target.setPose(numpy_to_robodk_mat(T_base_target))

    return target


def create_point_marker(rdk, name, position_base):
    T_base_target = np.eye(4, dtype=np.float64)
    T_base_target[:3, 3] = position_base

    return create_target_marker(
        rdk,
        name,
        T_base_target
    )


def create_debug_targets(rdk, targets):
    if not CREATE_DEBUG_TARGETS:
        return

    for index, (_, T_base_tcp, seam_point_base) in enumerate(targets, start=1):
        create_target_marker(
            rdk,
            f"ANGLED_TCP_TARGET_{index:02d}",
            T_base_tcp
        )

        create_point_marker(
            rdk,
            f"ANGLED_SEAM_POINT_{index:02d}",
            seam_point_base
        )


# ─────────────────────────────────────────────────────────────────────────────
# MAIN
# ─────────────────────────────────────────────────────────────────────────────

def main():
    rdk = Robolink()

    robot = rdk.ItemUserPick(
        "Select your Doosan M0609 robot",
        ITEM_TYPE_ROBOT
    )

    if not robot.Valid():
        raise Exception("No valid robot selected.")

    print("Selected robot:", robot.Name())

    connect_robot(robot, rdk)

    T_tcp_mount = xyzrxryrz_to_numpy(TCP_TO_CAMERA_MOUNT)
    T_mount_optical = xyzrxryrz_to_numpy(CAMERA_MOUNT_TO_OPTICAL)

    T_tcp_camera = T_tcp_mount @ T_mount_optical

    print_transform("T_tcp_camera", T_tcp_camera)

    try:
        move_robot_to_joints(
            robot,
            rdk,
            HOME_JOINTS,
            "Home_Start"
        )

        actual_center_joints = move_robot_to_joints(
            robot,
            rdk,
            CENTER_REFERENCE_JOINTS,
            "Center_Reference_View"
        )

        locked_j6_value = actual_center_joints[5]

        T_base_tcp_center = robodk_mat_to_numpy(
            robot.SolveFK(actual_center_joints)
        )

        T_base_camera_center = T_base_tcp_center @ T_tcp_camera

        print_transform("T_base_tcp_center", T_base_tcp_center)
        print_transform("T_base_camera_center", T_base_camera_center)
        print("")
        print("J6 reference value:", round(locked_j6_value, 2))

        seam_points_camera = generate_seam_points_camera_frame()

        seam_points_base = transform_seam_points_to_base(
            T_base_camera_center,
            seam_points_camera
        )

        targets = generate_angled_tcp_targets(
            T_base_camera_center,
            seam_points_base
        )

        create_debug_targets(
            rdk,
            targets
        )

        print("")
        print("=" * 70)
        print("ANGLED TIP PATH START")
        print("=" * 70)
        print("The tool now has an angle toward the seam.")
        print("The TCP is placed slightly before the seam using TIP_STANDOFF_M.")
        print("No welding machine or arc is triggered.")
        print("=" * 70)

        successful_moves = 0
        skipped_moves = 0
        failed_moves = 0

        seed_joints = actual_center_joints

        for label, T_base_tcp_target, seam_point_base in targets:
            if not is_pose_safe(
                T_base_tcp_target,
                label
            ):
                skipped_moves += 1
                continue

            try:
                actual_joints = move_robot_to_pose(
                    robot,
                    rdk,
                    T_base_tcp_target,
                    seed_joints,
                    locked_j6_value,
                    label
                )

                if LOCK_J6_WITH_SEED:
                    actual_joints[5] = locked_j6_value

                seed_joints = actual_joints

                successful_moves += 1

            except Exception as error:
                print("")
                print(f"WARNING: Could not move to {label}.")
                print("Move error:", error)
                failed_moves += 1
                continue

        print("")
        print("=" * 70)
        print("ANGLED TIP PATH FINISHED")
        print("=" * 70)
        print("Successful moves:", successful_moves)
        print("Skipped moves:", skipped_moves)
        print("Failed moves:", failed_moves)

    except KeyboardInterrupt:
        print("")
        print("Movement interrupted by user.")

    finally:
        try:
            move_robot_to_joints(
                robot,
                rdk,
                HOME_JOINTS,
                "Home_End"
            )
        except Exception as error:
            print("Could not move robot back to home position:", error)

    print("Done.")


if __name__ == "__main__":
    main()

--- Python program Prog5 ---
import sys
import time
from pathlib import Path

import cv2
import numpy as np
import open3d as o3d
import pyrealsense2 as rs

sys.path.append("C:/RoboDK/Python")

from robodk.robolink import *
from robodk.robomath import TxyzRxyz_2_Pose, Mat


# ─────────────────────────────────────────────────────────────────────────────
# CONFIGURATION
# ─────────────────────────────────────────────────────────────────────────────

RUN_ON_REAL_ROBOT = True

HOME_JOINTS = [270.00, 0.00, 90.00, 180.00, 0.00, 0.00]

CENTER_REFERENCE_JOINTS = [270.01, 0.21, 98.95, 180.00, 6.92, 0.00]

TCP_TO_CAMERA_MOUNT = [0, 0, 55, 0, 0, 0]
CAMERA_MOUNT_TO_OPTICAL = [0, 0, 0, 0, 0, 90]

MIN_SAFE_TCP_Z_MM = 120.0
MIN_SAFE_CAMERA_Z_MM = 120.0

RS_WIDTH = 848
RS_HEIGHT = 480
RS_FPS = 30

WARMUP_FRAMES = 30
CAPTURE_FRAMES_PER_POSITION = 30

DEPTH_TRUNC_MAX = 1.0

SETTLE_TIME = 1.5
MOVE_TIMEOUT_SEC = 30.0
POLL_INTERVAL_SEC = 0.1

SURFACE_VOXEL_SIZE = 0.003

OUTLIER_NB_NEIGHBORS = 20
OUTLIER_STD_RATIO = 2.0

NORMAL_RADIUS = 0.02
NORMAL_MAX_NN = 30

SHOW_FINAL_CLOUD = True
SHOW_DEBUG_EACH_SCAN = False

MIN_SIDE_OFFSET_M = 0.08
MAX_SIDE_OFFSET_M = 0.32

MIN_VERTICAL_OFFSET_M = 0.06
MAX_VERTICAL_OFFSET_M = 0.24

MIN_FORWARD_OFFSET_M = 0.03
MAX_FORWARD_OFFSET_M = 0.14

ADAPTIVE_CROP_MARGIN_X_M = 0.12
ADAPTIVE_CROP_MARGIN_Y_M = 0.12
ADAPTIVE_CROP_MARGIN_Z_M = 0.20

BOUNDS_LOW_PERCENTILE = 2.0
BOUNDS_HIGH_PERCENTILE = 98.0

MIN_REFERENCE_POINTS = 1000

OUTPUT_FOLDER = Path(
    "C:/Users/daryl/Desktop/Robotic D Environment Mapping/"
    "Robotic-3D-Environment-Mapping/Point Cloud Testing Folder"
)

OUTPUT_CLEAN_FILE = OUTPUT_FOLDER / "adaptive_inside_box_pointcloud_clean.pcd"


# ─────────────────────────────────────────────────────────────────────────────
# AUTO-CENTER CONFIGURATION
# ─────────────────────────────────────────────────────────────────────────────

AUTO_CENTER_BEFORE_SCAN = True
AUTO_CENTER_TARGET_DISTANCE_M = 0.80
AUTO_CENTER_MIN_DEPTH_M = 0.20
AUTO_CENTER_MAX_DEPTH_M = 3.00

AUTO_CENTER_MAX_TRANSLATION_STEP_M = 0.025
AUTO_CENTERING_GAIN = 0.60
AUTO_DEPTH_GAIN = 0.60

AUTO_CENTER_TOLERANCE_PX = 25
AUTO_DISTANCE_TOLERANCE_M = 0.05

AUTO_REQUIRED_STABLE_FRAMES = 8
AUTO_STABLE_CENTER_TOLERANCE_PX = 12
AUTO_STABLE_DISTANCE_TOLERANCE_M = 0.04
AUTO_MOVE_COOLDOWN_SECONDS = 1.25
AUTO_MAX_FAILED_MOVES = 5
AUTO_MAX_TOTAL_MOVES = 30
AUTO_CENTER_TIMEOUT_SECONDS = 180.0

AUTO_MIN_BOX_AREA = 1200
AUTO_MIN_BOX_WIDTH = 80
AUTO_MIN_BOX_HEIGHT = 80

AUTO_DEPTH_PERCENTILE = 10
AUTO_DEPTH_FRONT_MARGIN = 0.05
AUTO_DEPTH_BACK_MARGIN = 0.45

AUTO_DETECTION_ROI_TOP_RATIO = 0.05
AUTO_DETECTION_ROI_BOTTOM_RATIO = 0.82
AUTO_DETECTION_ROI_LEFT_RATIO = 0.02
AUTO_DETECTION_ROI_RIGHT_RATIO = 0.98

AUTO_WINDOW_NAME = "Automatic Box Centering"
AUTO_MASK_WINDOW_NAME = "Automatic Depth Mask"


# ─────────────────────────────────────────────────────────────────────────────
# ROBODK MATRIX HELPERS
# ─────────────────────────────────────────────────────────────────────────────

def robodk_mat_to_numpy(mat):
    transform = np.eye(4, dtype=np.float64)

    for row in range(3):
        for col in range(3):
            transform[row, col] = mat[row, col]

        transform[row, 3] = mat[row, 3] / 1000.0

    return transform


def numpy_to_robodk_mat(transform):
    return Mat([
        [
            transform[0, 0],
            transform[0, 1],
            transform[0, 2],
            transform[0, 3] * 1000.0,
        ],
        [
            transform[1, 0],
            transform[1, 1],
            transform[1, 2],
            transform[1, 3] * 1000.0,
        ],
        [
            transform[2, 0],
            transform[2, 1],
            transform[2, 2],
            transform[2, 3] * 1000.0,
        ],
        [0, 0, 0, 1],
    ])


def xyzrxryrz_to_numpy(pose_values):
    pose = TxyzRxyz_2_Pose([
        pose_values[0],
        pose_values[1],
        pose_values[2],
        np.radians(pose_values[3]),
        np.radians(pose_values[4]),
        np.radians(pose_values[5]),
    ])

    return robodk_mat_to_numpy(pose)


def make_local_offset_transform(offset_x, offset_y, offset_z):
    transform = np.eye(4, dtype=np.float64)
    transform[0, 3] = offset_x
    transform[1, 3] = offset_y
    transform[2, 3] = offset_z
    return transform


def joints_to_list(joints_mat):
    try:
        return list(joints_mat.list())
    except Exception:
        try:
            return list(joints_mat)
        except Exception:
            return [joints_mat[index] for index in range(len(joints_mat))]


def clamp(value, minimum_value, maximum_value):
    return max(minimum_value, min(value, maximum_value))


# ─────────────────────────────────────────────────────────────────────────────
# ROBODK ROBOT HELPERS
# ─────────────────────────────────────────────────────────────────────────────

def connect_robot(robot, rdk):
    if RUN_ON_REAL_ROBOT:
        rdk.setRunMode(RUNMODE_RUN_ROBOT)

        status = robot.ConnectSafe()
        print("ConnectSafe status:", status)

        if status != ROBOTCOM_READY:
            raise Exception("Robot is not ready. Check RoboDK connection settings.")
    else:
        rdk.setRunMode(RUNMODE_SIMULATE)
        print("Running in RoboDK simulation mode.")


def wait_until_robot_stops(robot, timeout_sec=MOVE_TIMEOUT_SEC):
    start = time.time()

    while True:
        try:
            if not robot.Busy():
                return
        except Exception:
            pass

        if time.time() - start > timeout_sec:
            raise Exception("Timeout waiting for robot to stop.")

        time.sleep(POLL_INTERVAL_SEC)


def get_robot_joints_when_ready(robot, timeout_sec=5.0):
    start = time.time()

    while True:
        try:
            return joints_to_list(robot.Joints())
        except Exception:
            if time.time() - start > timeout_sec:
                raise Exception("Could not read robot joints.")

            time.sleep(POLL_INTERVAL_SEC)


def move_robot_to_joints(robot, rdk, joints, label):
    target = rdk.AddTarget(f"_adaptive_inside_box_{label}")
    target.setAsJointTarget()
    target.setJoints(joints)

    print(f"\nMoving to {label}: {[round(joint, 2) for joint in joints]}")

    if RUN_ON_REAL_ROBOT:
        rdk.setRunMode(RUNMODE_RUN_ROBOT)
    else:
        rdk.setRunMode(RUNMODE_SIMULATE)

    robot.MoveJ(target, blocking=False)

    wait_until_robot_stops(robot)

    target.Delete()

    print(f"Arrived at {label}. Settling for {SETTLE_TIME:.1f} seconds...")
    time.sleep(SETTLE_TIME)

    return get_robot_joints_when_ready(robot)


def move_robot_to_pose(robot, rdk, T_base_tcp, label):
    target = rdk.AddTarget(f"_adaptive_inside_box_{label}")
    target_pose = numpy_to_robodk_mat(T_base_tcp)

    target.setPose(target_pose)
    target.setAsCartesianTarget()

    print(f"\nMoving to generated pose: {label}")
    print("Target TCP position in robot base frame:")
    print(f"X: {T_base_tcp[0, 3] * 1000.0:.1f} mm")
    print(f"Y: {T_base_tcp[1, 3] * 1000.0:.1f} mm")
    print(f"Z: {T_base_tcp[2, 3] * 1000.0:.1f} mm")

    if RUN_ON_REAL_ROBOT:
        rdk.setRunMode(RUNMODE_RUN_ROBOT)
    else:
        rdk.setRunMode(RUNMODE_SIMULATE)

    robot.MoveJ(target, blocking=False)

    wait_until_robot_stops(robot)

    target.Delete()

    print(f"Arrived at {label}. Settling for {SETTLE_TIME:.1f} seconds...")
    time.sleep(SETTLE_TIME)

    return get_robot_joints_when_ready(robot)


def is_generated_pose_safe(T_base_tcp, T_base_camera, label):
    tcp_z_mm = T_base_tcp[2, 3] * 1000.0
    camera_z_mm = T_base_camera[2, 3] * 1000.0

    if tcp_z_mm < MIN_SAFE_TCP_Z_MM:
        print("")
        print(f"SKIPPING {label}")
        print(f"Reason: TCP Z is too low: {tcp_z_mm:.1f} mm")
        print(f"Minimum safe TCP Z: {MIN_SAFE_TCP_Z_MM:.1f} mm")
        return False

    if camera_z_mm < MIN_SAFE_CAMERA_Z_MM:
        print("")
        print(f"SKIPPING {label}")
        print(f"Reason: Camera Z is too low: {camera_z_mm:.1f} mm")
        print(f"Minimum safe camera Z: {MIN_SAFE_CAMERA_Z_MM:.1f} mm")
        return False

    return True


def print_transform(name, transform):
    print(f"\n{name}:")
    print(np.round(transform, 6))


def print_cloud_bounds(name, point_cloud):
    if len(point_cloud.points) == 0:
        print(f"{name}: empty point cloud")
        return

    bounding_box = point_cloud.get_axis_aligned_bounding_box()

    print("")
    print(name)
    print("Points:", len(point_cloud.points))
    print("Min bound:", np.round(bounding_box.get_min_bound(), 4))
    print("Max bound:", np.round(bounding_box.get_max_bound(), 4))
    print("Center   :", np.round(bounding_box.get_center(), 4))
    print("Extent   :", np.round(bounding_box.get_extent(), 4))


# ─────────────────────────────────────────────────────────────────────────────
# REALSENSE HELPERS
# ─────────────────────────────────────────────────────────────────────────────

def start_realsense():
    print("\nStarting Intel RealSense D455f...")

    pipeline = rs.pipeline()
    config = rs.config()

    config.enable_stream(rs.stream.depth, RS_WIDTH, RS_HEIGHT, rs.format.z16, RS_FPS)
    config.enable_stream(rs.stream.color, RS_WIDTH, RS_HEIGHT, rs.format.rgb8, RS_FPS)

    profile = pipeline.start(config)

    depth_sensor = profile.get_device().first_depth_sensor()

    if depth_sensor.supports(rs.option.visual_preset):
        try:
            depth_sensor.set_option(
                rs.option.visual_preset,
                int(rs.rs400_visual_preset.high_density)
            )
            print("Visual preset: HIGH_DENSITY")
        except Exception as error:
            print("Could not set HIGH_DENSITY preset:", error)

    if depth_sensor.supports(rs.option.emitter_enabled):
        try:
            depth_sensor.set_option(rs.option.emitter_enabled, 1)
            print("Emitter enabled.")
        except Exception as error:
            print("Could not enable emitter:", error)

    if depth_sensor.supports(rs.option.laser_power):
        try:
            laser_range = depth_sensor.get_option_range(rs.option.laser_power)
            depth_sensor.set_option(rs.option.laser_power, laser_range.max)
            print("Laser power set to max:", laser_range.max)
        except Exception as error:
            print("Could not set laser power:", error)

    depth_scale = depth_sensor.get_depth_scale()
    print("Depth scale:", depth_scale)

    spatial_filter = rs.spatial_filter()
    temporal_filter = rs.temporal_filter()
    hole_filling_filter = rs.hole_filling_filter()

    spatial_filter.set_option(rs.option.filter_magnitude, 2)
    spatial_filter.set_option(rs.option.filter_smooth_alpha, 0.5)
    spatial_filter.set_option(rs.option.filter_smooth_delta, 20)

    hole_filling_filter.set_option(rs.option.holes_fill, 1)

    align = rs.align(rs.stream.color)

    print(f"Warming up RealSense for {WARMUP_FRAMES} frames...")
    for _ in range(WARMUP_FRAMES):
        pipeline.wait_for_frames()

    color_stream = profile.get_stream(rs.stream.color).as_video_stream_profile()
    intrinsics = color_stream.get_intrinsics()

    intrinsic_o3d = o3d.camera.PinholeCameraIntrinsic(
        intrinsics.width,
        intrinsics.height,
        intrinsics.fx,
        intrinsics.fy,
        intrinsics.ppx,
        intrinsics.ppy,
    )

    print(f"RealSense ready: fx={intrinsics.fx:.1f}, fy={intrinsics.fy:.1f}")

    return (
        pipeline,
        align,
        depth_scale,
        intrinsic_o3d,
        spatial_filter,
        temporal_filter,
        hole_filling_filter,
    )


def make_rgbd(color_image, depth_image, depth_scale_value):
    color_o3d = o3d.geometry.Image(color_image.astype(np.uint8))
    depth_o3d = o3d.geometry.Image(depth_image.astype(np.uint16))

    return o3d.geometry.RGBDImage.create_from_color_and_depth(
        color_o3d,
        depth_o3d,
        depth_scale=1.0 / depth_scale_value,
        depth_trunc=DEPTH_TRUNC_MAX,
        convert_rgb_to_intensity=False,
    )


def capture_stable_pointcloud(
    pipeline,
    align,
    intrinsic_o3d,
    depth_scale_value,
    spatial_filter,
    temporal_filter,
    hole_filling_filter,
    frames_to_capture=CAPTURE_FRAMES_PER_POSITION
):
    color_stack = []
    depth_stack = []

    print(f"Capturing {frames_to_capture} frames...")

    for frame_index in range(frames_to_capture):
        frames = pipeline.wait_for_frames()
        aligned_frames = align.process(frames)

        depth_frame = aligned_frames.get_depth_frame()
        color_frame = aligned_frames.get_color_frame()

        if not depth_frame or not color_frame:
            print(f"Frame {frame_index + 1}: skipped because depth or color is missing.")
            continue

        depth_frame = spatial_filter.process(depth_frame)
        depth_frame = temporal_filter.process(depth_frame)
        depth_frame = hole_filling_filter.process(depth_frame)

        depth_stack.append(np.asanyarray(depth_frame.get_data()).astype(np.uint16))
        color_stack.append(np.asanyarray(color_frame.get_data()).astype(np.uint8))

        print(f"Frame {frame_index + 1}/{frames_to_capture} captured.")

    if not depth_stack:
        return None

    print("Combining frames into one stable point cloud...")

    depth_median = np.median(np.stack(depth_stack, axis=0), axis=0).astype(np.uint16)
    color_mean = np.mean(np.stack(color_stack, axis=0), axis=0).astype(np.uint8)

    rgbd = make_rgbd(color_mean, depth_median, depth_scale_value)

    point_cloud = o3d.geometry.PointCloud.create_from_rgbd_image(
        rgbd,
        intrinsic_o3d,
    )

    if len(point_cloud.points) == 0:
        return None

    return point_cloud


# ─────────────────────────────────────────────────────────────────────────────
# ADAPTIVE POINT CLOUD HELPERS
# ─────────────────────────────────────────────────────────────────────────────

def estimate_camera_cloud_bounds(point_cloud):
    points = np.asarray(point_cloud.points)

    if len(points) < MIN_REFERENCE_POINTS:
        raise Exception(
            f"Not enough points for adaptive scan estimation. "
            f"Points found: {len(points)}"
        )

    valid_mask = (
        np.isfinite(points[:, 0]) &
        np.isfinite(points[:, 1]) &
        np.isfinite(points[:, 2]) &
        (points[:, 2] > 0.05) &
        (points[:, 2] < DEPTH_TRUNC_MAX)
    )

    points = points[valid_mask]

    if len(points) < MIN_REFERENCE_POINTS:
        raise Exception(
            f"Not enough valid depth points for adaptive scan estimation. "
            f"Valid points found: {len(points)}"
        )

    min_x = np.percentile(points[:, 0], BOUNDS_LOW_PERCENTILE)
    max_x = np.percentile(points[:, 0], BOUNDS_HIGH_PERCENTILE)

    min_y = np.percentile(points[:, 1], BOUNDS_LOW_PERCENTILE)
    max_y = np.percentile(points[:, 1], BOUNDS_HIGH_PERCENTILE)

    min_z = np.percentile(points[:, 2], BOUNDS_LOW_PERCENTILE)
    max_z = np.percentile(points[:, 2], BOUNDS_HIGH_PERCENTILE)

    center_x = float((min_x + max_x) / 2.0)
    center_y = float((min_y + max_y) / 2.0)
    center_z = float(np.median(points[:, 2]))

    extent_x = float(max_x - min_x)
    extent_y = float(max_y - min_y)
    extent_z = float(max_z - min_z)

    bounds = {
        "min_x": float(min_x),
        "max_x": float(max_x),
        "min_y": float(min_y),
        "max_y": float(max_y),
        "min_z": float(min_z),
        "max_z": float(max_z),
        "center_x": center_x,
        "center_y": center_y,
        "center_z": center_z,
        "extent_x": extent_x,
        "extent_y": extent_y,
        "extent_z": extent_z,
    }

    print("")
    print("Adaptive camera-frame bounds estimated from reference scan:")
    for key, value in bounds.items():
        print(f"{key}: {value:.4f} m")

    return bounds


def crop_pointcloud_adaptive(point_cloud, adaptive_bounds):
    if len(point_cloud.points) == 0:
        return point_cloud

    points = np.asarray(point_cloud.points)

    min_x = adaptive_bounds["min_x"] - ADAPTIVE_CROP_MARGIN_X_M
    max_x = adaptive_bounds["max_x"] + ADAPTIVE_CROP_MARGIN_X_M

    min_y = adaptive_bounds["min_y"] - ADAPTIVE_CROP_MARGIN_Y_M
    max_y = adaptive_bounds["max_y"] + ADAPTIVE_CROP_MARGIN_Y_M

    min_z = max(0.05, adaptive_bounds["min_z"] - ADAPTIVE_CROP_MARGIN_Z_M)
    max_z = min(DEPTH_TRUNC_MAX, adaptive_bounds["max_z"] + ADAPTIVE_CROP_MARGIN_Z_M)

    mask = (
        (points[:, 0] >= min_x) &
        (points[:, 0] <= max_x) &
        (points[:, 1] >= min_y) &
        (points[:, 1] <= max_y) &
        (points[:, 2] >= min_z) &
        (points[:, 2] <= max_z)
    )

    indices = np.where(mask)[0]

    if len(indices) == 0:
        print("WARNING: Adaptive crop removed all points. Keeping original cloud.")
        return point_cloud

    cropped_cloud = point_cloud.select_by_index(indices)

    print("Adaptive camera-frame crop enabled.")
    print("Points before adaptive crop:", len(point_cloud.points))
    print("Points after adaptive crop :", len(cropped_cloud.points))

    return cropped_cloud


def clean_pointcloud(point_cloud):
    if len(point_cloud.points) == 0:
        return point_cloud

    point_cloud = point_cloud.voxel_down_sample(voxel_size=SURFACE_VOXEL_SIZE)

    if len(point_cloud.points) == 0:
        return point_cloud

    point_cloud, _ = point_cloud.remove_statistical_outlier(
        nb_neighbors=OUTLIER_NB_NEIGHBORS,
        std_ratio=OUTLIER_STD_RATIO,
    )

    return point_cloud


def estimate_normals(point_cloud):
    if len(point_cloud.points) == 0:
        return point_cloud

    point_cloud.estimate_normals(
        search_param=o3d.geometry.KDTreeSearchParamHybrid(
            radius=NORMAL_RADIUS,
            max_nn=NORMAL_MAX_NN,
        )
    )

    return point_cloud


def save_debug_scan(label, point_cloud):
    debug_file = OUTPUT_FOLDER / f"debug_{label}.pcd"

    o3d.io.write_point_cloud(str(debug_file), point_cloud)

    print("Saved debug scan:", debug_file)
    print_cloud_bounds(f"Debug scan bounds - {label}", point_cloud)


# ─────────────────────────────────────────────────────────────────────────────
# ADAPTIVE SCAN POSE GENERATION
# ─────────────────────────────────────────────────────────────────────────────

def generate_adaptive_scan_offsets(adaptive_bounds):
    extent_x = adaptive_bounds["extent_x"]
    extent_y = adaptive_bounds["extent_y"]

    center_x = adaptive_bounds["center_x"]
    center_y = adaptive_bounds["center_y"]
    center_z = adaptive_bounds["center_z"]

    side_offset = clamp(
        extent_x * 0.35,
        MIN_SIDE_OFFSET_M,
        MAX_SIDE_OFFSET_M,
    )

    vertical_offset = clamp(
        extent_y * 0.35,
        MIN_VERTICAL_OFFSET_M,
        MAX_VERTICAL_OFFSET_M,
    )

    forward_offset = clamp(
        center_z * 0.12,
        MIN_FORWARD_OFFSET_M,
        MAX_FORWARD_OFFSET_M,
    )

    print("")
    print("Adaptive scan movement offsets:")
    print(f"Side offset: {side_offset:.4f} m")
    print(f"Vertical offset: {vertical_offset:.4f} m")
    print(f"Forward offset: {forward_offset:.4f} m")

    return [
        ("Reference_Center", 0.00, 0.00, 0.00),

        ("Left_Inside_Area", center_x - side_offset, center_y, 0.00),
        ("Right_Inside_Area", center_x + side_offset, center_y, 0.00),

        ("Upper_Inside_Area", center_x, center_y - vertical_offset, 0.00),
        ("Lower_Inside_Area", center_x, center_y + vertical_offset, 0.00),

        ("Upper_Left_Inside_Area", center_x - side_offset, center_y - vertical_offset, 0.00),
        ("Upper_Right_Inside_Area", center_x + side_offset, center_y - vertical_offset, 0.00),

        ("Lower_Left_Inside_Area", center_x - side_offset, center_y + vertical_offset, 0.00),
        ("Lower_Right_Inside_Area", center_x + side_offset, center_y + vertical_offset, 0.00),

        ("Closer_Center", center_x, center_y, forward_offset),
        ("Closer_Left", center_x - side_offset * 0.70, center_y, forward_offset),
        ("Closer_Right", center_x + side_offset * 0.70, center_y, forward_offset),
        ("Closer_Upper", center_x, center_y - vertical_offset * 0.70, forward_offset),
        ("Closer_Lower", center_x, center_y + vertical_offset * 0.70, forward_offset),
    ]


def generate_scan_camera_poses_from_center(T_base_camera_center, adaptive_bounds):
    generated_poses = []

    adaptive_offsets = generate_adaptive_scan_offsets(adaptive_bounds)

    print("\nGenerating adaptive scan poses from center reference...")
    print("Center camera position in robot base frame:")
    print(f"X: {T_base_camera_center[0, 3] * 1000.0:.1f} mm")
    print(f"Y: {T_base_camera_center[1, 3] * 1000.0:.1f} mm")
    print(f"Z: {T_base_camera_center[2, 3] * 1000.0:.1f} mm")

    for label, offset_x, offset_y, offset_z in adaptive_offsets:
        T_camera_offset = make_local_offset_transform(
            offset_x,
            offset_y,
            offset_z,
        )

        T_base_camera_target = T_base_camera_center @ T_camera_offset

        print("")
        print(f"Generated camera pose: {label}")
        print(f"Local offset X: {offset_x * 1000.0:.1f} mm")
        print(f"Local offset Y: {offset_y * 1000.0:.1f} mm")
        print(f"Local offset Z: {offset_z * 1000.0:.1f} mm")
        print("Generated camera position in robot base frame:")
        print(f"X: {T_base_camera_target[0, 3] * 1000.0:.1f} mm")
        print(f"Y: {T_base_camera_target[1, 3] * 1000.0:.1f} mm")
        print(f"Z: {T_base_camera_target[2, 3] * 1000.0:.1f} mm")

        generated_poses.append((label, T_base_camera_target))

    return generated_poses


# ─────────────────────────────────────────────────────────────────────────────
# SCANNING LOGIC
# ─────────────────────────────────────────────────────────────────────────────

def scan_current_position(
    label,
    pipeline,
    align,
    intrinsic_o3d,
    depth_scale,
    spatial_filter,
    temporal_filter,
    hole_filling_filter,
    T_base_camera_actual,
    adaptive_bounds=None,
):
    point_cloud = capture_stable_pointcloud(
        pipeline,
        align,
        intrinsic_o3d,
        depth_scale,
        spatial_filter,
        temporal_filter,
        hole_filling_filter,
        CAPTURE_FRAMES_PER_POSITION,
    )

    if point_cloud is None:
        print(f"WARNING: Empty point cloud at {label}.")
        return None

    print(f"Captured raw camera points at {label}: {len(point_cloud.points):,}")
    print_cloud_bounds(f"Raw camera-frame scan - {label}", point_cloud)

    if adaptive_bounds is not None:
        point_cloud = crop_pointcloud_adaptive(point_cloud, adaptive_bounds)

    if len(point_cloud.points) == 0:
        print(f"WARNING: Empty point cloud after adaptive crop at {label}.")
        return None

    print_cloud_bounds(f"Cropped camera-frame scan - {label}", point_cloud)

    point_cloud.transform(T_base_camera_actual)

    clean_scan = clean_pointcloud(point_cloud)

    if len(clean_scan.points) == 0:
        print(f"WARNING: Point cloud empty after cleaning at {label}.")
        return None

    save_debug_scan(label, clean_scan)

    if SHOW_DEBUG_EACH_SCAN:
        o3d.visualization.draw_geometries(
            [clean_scan],
            window_name=f"Debug transformed scan - {label}",
        )

    return clean_scan



# ─────────────────────────────────────────────────────────────────────────────
# AUTO-CENTERING HELPERS
# ─────────────────────────────────────────────────────────────────────────────

def get_aligned_realsense_frame(pipeline, align):
    frames = pipeline.wait_for_frames()
    aligned_frames = align.process(frames)

    depth_frame = aligned_frames.get_depth_frame()
    color_frame = aligned_frames.get_color_frame()

    if not depth_frame or not color_frame:
        return None, None, None

    depth_image = np.asanyarray(depth_frame.get_data())
    color_image_rgb = np.asanyarray(color_frame.get_data())

    return depth_frame, color_image_rgb, depth_image


def get_auto_depth_in_region(depth_image, depth_scale, x1, y1, x2, y2):
    image_height, image_width = depth_image.shape

    x1 = max(0, min(int(x1), image_width))
    x2 = max(0, min(int(x2), image_width))
    y1 = max(0, min(int(y1), image_height))
    y2 = max(0, min(int(y2), image_height))

    if x2 <= x1 or y2 <= y1:
        return None

    depth_crop = depth_image[y1:y2, x1:x2].astype(np.float32) * depth_scale

    valid_depth = depth_crop[
        (depth_crop > AUTO_CENTER_MIN_DEPTH_M)
        & (depth_crop < AUTO_CENTER_MAX_DEPTH_M)
    ]

    if valid_depth.size == 0:
        return None

    return float(np.percentile(valid_depth, 30))


def create_auto_detection_roi_mask(image_height, image_width):
    roi_mask = np.zeros((image_height, image_width), dtype=np.uint8)

    x1 = int(image_width * AUTO_DETECTION_ROI_LEFT_RATIO)
    x2 = int(image_width * AUTO_DETECTION_ROI_RIGHT_RATIO)
    y1 = int(image_height * AUTO_DETECTION_ROI_TOP_RATIO)
    y2 = int(image_height * AUTO_DETECTION_ROI_BOTTOM_RATIO)

    roi_mask[y1:y2, x1:x2] = 255

    return roi_mask


def create_auto_depth_mask(depth_image, depth_scale):
    image_height, image_width = depth_image.shape
    depth_meters = depth_image.astype(np.float32) * depth_scale

    roi_mask = create_auto_detection_roi_mask(image_height, image_width)

    valid_mask = (
        (depth_meters > AUTO_CENTER_MIN_DEPTH_M)
        & (depth_meters < AUTO_CENTER_MAX_DEPTH_M)
        & (roi_mask == 255)
    )

    if not np.any(valid_mask):
        return None

    valid_depth_values = depth_meters[valid_mask]
    front_depth = np.percentile(valid_depth_values, AUTO_DEPTH_PERCENTILE)

    mask = (
        valid_mask
        & (depth_meters > front_depth - AUTO_DEPTH_FRONT_MARGIN)
        & (depth_meters < front_depth + AUTO_DEPTH_BACK_MARGIN)
    )

    mask = mask.astype(np.uint8) * 255

    close_kernel = np.ones((11, 11), np.uint8)
    open_kernel = np.ones((5, 5), np.uint8)

    mask = cv2.morphologyEx(mask, cv2.MORPH_CLOSE, close_kernel, iterations=3)
    mask = cv2.morphologyEx(mask, cv2.MORPH_OPEN, open_kernel, iterations=1)
    mask = cv2.bitwise_and(mask, roi_mask)

    return mask


def detect_auto_box(depth_image, depth_scale):
    mask = create_auto_depth_mask(depth_image, depth_scale)

    if mask is None:
        return None, None

    contours, _ = cv2.findContours(
        mask,
        cv2.RETR_EXTERNAL,
        cv2.CHAIN_APPROX_SIMPLE,
    )

    image_height, image_width = depth_image.shape
    image_center_x = image_width / 2.0
    image_center_y = image_height / 2.0

    best_box = None
    best_score = 0

    for contour in contours:
        area = cv2.contourArea(contour)

        if area < AUTO_MIN_BOX_AREA:
            continue

        x, y, width, height = cv2.boundingRect(contour)

        if width < AUTO_MIN_BOX_WIDTH or height < AUTO_MIN_BOX_HEIGHT:
            continue

        if width > image_width * 0.98 or height > image_height * 0.98:
            continue

        aspect_ratio = width / float(height)

        if aspect_ratio < 0.50 or aspect_ratio > 4.50:
            continue

        x1 = x
        y1 = y
        x2 = x + width
        y2 = y + height

        center_x = int((x1 + x2) / 2)
        center_y = int((y1 + y2) / 2)

        distance_meters = get_auto_depth_in_region(
            depth_image,
            depth_scale,
            x1,
            y1,
            x2,
            y2,
        )

        if distance_meters is None:
            continue

        center_error = np.sqrt(
            (center_x - image_center_x) ** 2
            + (center_y - image_center_y) ** 2
        )

        area_score = area / float(image_width * image_height)
        center_score = 1.0 / (1.0 + center_error)
        score = area_score * 1000.0 + center_score * 150.0

        if score > best_score:
            best_score = score
            best_box = {
                "x1": x1,
                "y1": y1,
                "x2": x2,
                "y2": y2,
                "center_x": center_x,
                "center_y": center_y,
                "distance_meters": distance_meters,
                "area": area,
            }

    return best_box, mask


def get_auto_box_center_3d(depth_frame, box):
    center_x = box["center_x"]
    center_y = box["center_y"]
    depth_meters = box["distance_meters"]

    if depth_meters is None:
        return None

    if depth_meters <= AUTO_CENTER_MIN_DEPTH_M:
        return None

    if depth_meters >= AUTO_CENTER_MAX_DEPTH_M:
        return None

    intrinsics = depth_frame.profile.as_video_stream_profile().intrinsics

    point_camera = rs.rs2_deproject_pixel_to_point(
        intrinsics,
        [center_x, center_y],
        depth_meters,
    )

    return np.array(point_camera, dtype=np.float64)


def get_auto_box_offset_pixels(box):
    image_center_x = int(RS_WIDTH / 2)
    image_center_y = int(RS_HEIGHT / 2)

    offset_x = box["center_x"] - image_center_x
    offset_y = box["center_y"] - image_center_y

    return offset_x, offset_y


def is_auto_box_centered(box):
    offset_x, offset_y = get_auto_box_offset_pixels(box)

    center_error = np.sqrt(offset_x ** 2 + offset_y ** 2)
    distance_error = abs(box["distance_meters"] - AUTO_CENTER_TARGET_DISTANCE_M)

    return (
        center_error <= AUTO_CENTER_TOLERANCE_PX
        and distance_error <= AUTO_DISTANCE_TOLERANCE_M
    )


def is_auto_box_stable(current_box, previous_box):
    if current_box is None or previous_box is None:
        return False

    center_change = np.sqrt(
        (current_box["center_x"] - previous_box["center_x"]) ** 2
        + (current_box["center_y"] - previous_box["center_y"]) ** 2
    )

    distance_change = abs(
        current_box["distance_meters"] - previous_box["distance_meters"]
    )

    return (
        center_change <= AUTO_STABLE_CENTER_TOLERANCE_PX
        and distance_change <= AUTO_STABLE_DISTANCE_TOLERANCE_M
    )


def update_auto_stability(box, previous_box, stable_frame_count):
    if box is None:
        return 0, None

    if is_auto_box_stable(box, previous_box):
        stable_frame_count += 1
    else:
        stable_frame_count = 1

    return stable_frame_count, box


def calculate_auto_camera_correction(point_camera):
    camera_offset = np.array([
        point_camera[0] * AUTO_CENTERING_GAIN,
        point_camera[1] * AUTO_CENTERING_GAIN,
        (point_camera[2] - AUTO_CENTER_TARGET_DISTANCE_M) * AUTO_DEPTH_GAIN,
    ])

    offset_size = np.linalg.norm(camera_offset)

    if offset_size > AUTO_CENTER_MAX_TRANSLATION_STEP_M:
        camera_offset = (
            camera_offset / offset_size
        ) * AUTO_CENTER_MAX_TRANSLATION_STEP_M

    return camera_offset


def move_camera_one_auto_step_to_box_center(
    robot,
    rdk,
    T_tcp_camera,
    T_camera_tcp,
    point_camera,
):
    actual_joints = get_robot_joints_when_ready(robot)

    T_base_tcp_current = robodk_mat_to_numpy(robot.SolveFK(actual_joints))
    T_base_camera_current = T_base_tcp_current @ T_tcp_camera

    camera_offset = calculate_auto_camera_correction(point_camera)

    T_camera_offset = make_local_offset_transform(
        camera_offset[0],
        camera_offset[1],
        camera_offset[2],
    )

    T_base_camera_target = T_base_camera_current @ T_camera_offset
    T_base_tcp_target = T_base_camera_target @ T_camera_tcp

    print("")
    print("Automatic box-centering movement")
    print("3D box point in camera frame:", np.round(point_camera, 4), "m")
    print("Camera movement step:", np.round(camera_offset, 4), "m")
    print("Current robot joints:", [round(joint, 2) for joint in actual_joints])

    if not is_generated_pose_safe(
        T_base_tcp_target,
        T_base_camera_target,
        "Auto_Box_Center_Step",
    ):
        return None

    try:
        return move_robot_to_pose(
            robot,
            rdk,
            T_base_tcp_target,
            "Auto_Box_Center_Step",
        )
    except Exception as error:
        print("")
        print("Could not move robot to automatic box center step.")
        print("Move error:", error)
        return None


def should_auto_center_move(
    box,
    stable_frame_count,
    last_auto_move_time,
    failed_auto_moves,
    total_auto_moves,
):
    if box is None:
        return False

    if is_auto_box_centered(box):
        return False

    if stable_frame_count < AUTO_REQUIRED_STABLE_FRAMES:
        return False

    if time.time() - last_auto_move_time < AUTO_MOVE_COOLDOWN_SECONDS:
        return False

    if failed_auto_moves >= AUTO_MAX_FAILED_MOVES:
        return False

    if total_auto_moves >= AUTO_MAX_TOTAL_MOVES:
        return False

    return True


def draw_auto_box(image, box):
    image_center_x = int(RS_WIDTH / 2)
    image_center_y = int(RS_HEIGHT / 2)

    cv2.rectangle(
        image,
        (box["x1"], box["y1"]),
        (box["x2"], box["y2"]),
        (0, 255, 0),
        3,
    )

    cv2.circle(
        image,
        (box["center_x"], box["center_y"]),
        7,
        (0, 0, 255),
        -1,
    )

    cv2.line(
        image,
        (image_center_x - 15, image_center_y),
        (image_center_x + 15, image_center_y),
        (255, 0, 0),
        2,
    )

    cv2.line(
        image,
        (image_center_x, image_center_y - 15),
        (image_center_x, image_center_y + 15),
        (255, 0, 0),
        2,
    )

    cv2.line(
        image,
        (image_center_x, image_center_y),
        (box["center_x"], box["center_y"]),
        (0, 255, 255),
        2,
    )

    cv2.putText(
        image,
        f"Box | {box['distance_meters']:.2f} m",
        (box["x1"], max(box["y1"] - 10, 25)),
        cv2.FONT_HERSHEY_SIMPLEX,
        0.65,
        (0, 255, 0),
        2,
    )


def draw_auto_text(image, text, y, color):
    cv2.putText(
        image,
        text,
        (10, y),
        cv2.FONT_HERSHEY_SIMPLEX,
        0.65,
        color,
        2,
    )


